(* IEC 61131-3 sources: SmartHomeNew/ (part 4) *)

(* ---- FB_Cluster_Runtime_FSM.st ---- *)
FUNCTION_BLOCK FB_Cluster_Runtime_FSM
VAR_INPUT
    VI_Enable : BOOL;
    VI_System_Time_MS : UDINT;
END_VAR

IF NOT VI_Enable THEN
    GVL_Cluster_Runtime_FSM.G_Runtime_Valid := FALSE;
    RETURN;
END_IF;

// Reset runtime states.
GVL_Cluster_Runtime_FSM.G_State_Startup := FALSE;
GVL_Cluster_Runtime_FSM.G_State_Discovery := FALSE;
GVL_Cluster_Runtime_FSM.G_State_Synchronization := FALSE;
GVL_Cluster_Runtime_FSM.G_State_Operational := FALSE;
GVL_Cluster_Runtime_FSM.G_State_Degraded := FALSE;
GVL_Cluster_Runtime_FSM.G_State_Observer_Only := FALSE;
GVL_Cluster_Runtime_FSM.G_State_Recovery_Lock := FALSE;
GVL_Cluster_Runtime_FSM.G_State_Quarantine := FALSE;

// Startup state.
IF NOT GVL_Distributed_Runtime.G_Runtime_Valid THEN

    GVL_Cluster_Runtime_FSM.G_State_Startup := TRUE;

    GVL_Cluster_Runtime_FSM.G_Status_Code := 1;
    GVL_Cluster_Runtime_FSM.G_Status_Text :=
        'Cluster runtime startup';

ELSIF GVL_Runtime_Discovery.G_Runtime_Valid
   AND NOT GVL_Runtime_Discovery.G_Any_Discovery_Rejected THEN

    GVL_Cluster_Runtime_FSM.G_State_Discovery := TRUE;

    GVL_Cluster_Runtime_FSM.G_Status_Code := 2;
    GVL_Cluster_Runtime_FSM.G_Status_Text :=
        'Cluster runtime discovery';

END_IF;

// Synchronization state.
IF GVL_Runtime_Bus.G_TX_Healthy
   AND GVL_Runtime_Bus.G_RX_Healthy THEN

    GVL_Cluster_Runtime_FSM.G_State_Synchronization := TRUE;

END_IF;

// Operational state.
IF GVL_Distributed_Execution_Gates.G_Can_Execute
   AND GVL_Distributed_Execution_Gates.G_Can_Orchestrate THEN

    GVL_Cluster_Runtime_FSM.G_State_Operational := TRUE;

    GVL_Cluster_Runtime_FSM.G_Status_Code := 0;
    GVL_Cluster_Runtime_FSM.G_Status_Text :=
        'Cluster runtime operational';

END_IF;

// Degraded state.
IF GVL_Cluster_Safety_Barrier.G_Cluster_Execution_Blocked THEN

    GVL_Cluster_Runtime_FSM.G_State_Degraded := TRUE;

    GVL_Cluster_Runtime_FSM.G_Status_Code := 10;
    GVL_Cluster_Runtime_FSM.G_Status_Text :=
        'Cluster runtime degraded';

END_IF;

// Observer-only state.
IF GVL_Distributed_Authority.G_Authority_State.Authority_Observer_Only THEN

    GVL_Cluster_Runtime_FSM.G_State_Observer_Only := TRUE;

    GVL_Cluster_Runtime_FSM.G_Status_Code := 11;
    GVL_Cluster_Runtime_FSM.G_Status_Text :=
        'Cluster runtime observer-only';

END_IF;

// Recovery lock state.
IF GVL_Distributed_Recovery_Lock.G_Recovery_Execution_Blocked THEN

    GVL_Cluster_Runtime_FSM.G_State_Recovery_Lock := TRUE;

    GVL_Cluster_Runtime_FSM.G_Status_Code := 12;
    GVL_Cluster_Runtime_FSM.G_Status_Text :=
        'Cluster runtime recovery-locked';

END_IF;

// Quarantine state.
IF GVL_Runtime_Discovery.G_Any_Node_Quarantined THEN

    GVL_Cluster_Runtime_FSM.G_State_Quarantine := TRUE;

    GVL_Cluster_Runtime_FSM.G_Status_Code := 13;
    GVL_Cluster_Runtime_FSM.G_Status_Text :=
        'Cluster runtime quarantined';

END_IF;

GVL_Cluster_Runtime_FSM.G_Runtime_Valid := TRUE;
GVL_Cluster_Runtime_FSM.G_Last_Update_MS := VI_System_Time_MS;

END_FUNCTION_BLOCK

(* ---- FB_Cluster_Safety_Barrier_Runtime.st ---- *)
FUNCTION_BLOCK FB_Cluster_Safety_Barrier_Runtime
VAR_INPUT
    VI_Enable : BOOL;
    VI_System_Time_MS : UDINT;
END_VAR
VAR
    L_Block_Execution : BOOL;
    L_Status_Code : UINT;
    L_Status_Text : STRING(160);
END_VAR

IF NOT VI_Enable THEN
    GVL_Cluster_Safety_Barrier.G_Runtime_Valid := FALSE;
    RETURN;
END_IF;

L_Block_Execution := FALSE;
L_Status_Code := 0;
L_Status_Text := 'Cluster safety barrier healthy';

GVL_Cluster_Safety_Barrier.G_Remote_Authority_Degraded := FALSE;
GVL_Cluster_Safety_Barrier.G_Runtime_Bus_Degraded := FALSE;
GVL_Cluster_Safety_Barrier.G_Projection_Ownership_Invalid := FALSE;
GVL_Cluster_Safety_Barrier.G_Recovery_Lock_Active := FALSE;
GVL_Cluster_Safety_Barrier.G_Deployment_Invalid := FALSE;
GVL_Cluster_Safety_Barrier.G_Authority_Downgraded := FALSE;
GVL_Cluster_Safety_Barrier.G_Orchestration_Restricted := FALSE;

// Remote authority staleness barrier.
IF GVL_Distributed_Runtime.G_Any_Remote_Node_Offline
   OR GVL_Distributed_Runtime.G_Split_Brain_Suspected THEN

    L_Block_Execution := TRUE;
    L_Status_Code := 10;
    L_Status_Text :=
        'Cluster authority state degraded';

    GVL_Cluster_Safety_Barrier.G_Remote_Authority_Degraded := TRUE;

END_IF;

// Runtime bus integrity barrier.
IF GVL_Runtime_Bus.G_Any_Replication_Rejected
   OR NOT GVL_Runtime_Bus.G_TX_Healthy
   OR NOT GVL_Runtime_Bus.G_RX_Healthy THEN

    L_Block_Execution := TRUE;
    L_Status_Code := 11;
    L_Status_Text :=
        'Runtime bus integrity degraded';

    GVL_Cluster_Safety_Barrier.G_Runtime_Bus_Degraded := TRUE;

END_IF;

// Projection ownership barrier.
IF GVL_Distributed_Projection_Ownership.G_Any_Ownership_Conflict
   OR GVL_Distributed_Projection_Ownership.G_Any_Ownership_Stale THEN

    L_Block_Execution := TRUE;
    L_Status_Code := 12;
    L_Status_Text :=
        'Distributed projection ownership invalid';

    GVL_Cluster_Safety_Barrier.G_Projection_Ownership_Invalid := TRUE;

END_IF;

// Recovery lock barrier.
IF GVL_Distributed_Recovery_Lock.G_Recovery_Execution_Blocked
   OR GVL_Distributed_Recovery_Lock.G_Rollback_Execution_Blocked
   OR GVL_Distributed_Recovery_Lock.G_Reopen_Execution_Blocked THEN

    L_Block_Execution := TRUE;
    L_Status_Code := 13;
    L_Status_Text :=
        'Distributed recovery execution blocked';

    GVL_Cluster_Safety_Barrier.G_Recovery_Lock_Active := TRUE;

END_IF;

// Discovery/deployment barrier.
IF GVL_Runtime_Discovery.G_Any_Discovery_Rejected
   OR GVL_Runtime_Discovery.G_Any_Node_Quarantined THEN

    L_Block_Execution := TRUE;
    L_Status_Code := 14;
    L_Status_Text :=
        'Runtime deployment/discovery invalid';

    GVL_Cluster_Safety_Barrier.G_Deployment_Invalid := TRUE;

END_IF;

// Cluster escalation semantics.
IF L_Block_Execution THEN

    GVL_Distributed_Authority.G_Authority_State.Authority_Observer_Only := TRUE;
    GVL_Distributed_Authority.G_Authority_State.Authority_Master_Elected := FALSE;

    GVL_Distributed_Orchestration.G_Distributed_Projection_Healthy := FALSE;

    GVL_Cluster_Safety_Barrier.G_Authority_Downgraded := TRUE;
    GVL_Cluster_Safety_Barrier.G_Orchestration_Restricted := TRUE;

END_IF;

GVL_Cluster_Safety_Barrier.G_Cluster_Execution_Blocked :=
    L_Block_Execution;

GVL_Cluster_Safety_Barrier.G_Runtime_Valid := TRUE;
GVL_Cluster_Safety_Barrier.G_Last_Update_MS := VI_System_Time_MS;
GVL_Cluster_Safety_Barrier.G_Status_Code := L_Status_Code;
GVL_Cluster_Safety_Barrier.G_Status_Text := L_Status_Text;

END_FUNCTION_BLOCK

(* ---- FB_CO_Detector.st ---- *)
FUNCTION_BLOCK FB_CO_Detector
VAR_INPUT
    VI_CO_PPM : REAL;
    VI_Threshold_Warning : REAL := 30.0;
    VI_Threshold_Alarm   : REAL := 70.0;
END_VAR
VAR_OUTPUT
    VO_CO_Warning_Level : BOOL;
    VO_CO_Alarm_Level   : BOOL;
END_VAR

VO_CO_Warning_Level := (VI_CO_PPM >= VI_Threshold_Warning);
VO_CO_Alarm_Level   := (VI_CO_PPM >= VI_Threshold_Alarm);

(* ---- FB_Command_Deduplication.st ---- *)
FUNCTION_BLOCK FB_Command_Deduplication
VAR_INPUT
    VI_Command_ID : UDINT; // Unique ID from Gateway/HMI
    VI_Command_Type : E_Gateway_Command_Type;
    VI_Command_Value : REAL;
    VI_System_Time_MS : UDINT;
END_VAR
VAR_OUTPUT
    VO_Is_New_Command : BOOL; // TRUE if this command should be executed
    VO_Processed_ID : UDINT;
END_VAR
VAR
    L_Processed_History : ARRAY[0..GVL_CONSTANTS.C_MAX_DEDUPLICATION_HISTORY-1] OF UDINT;
    L_Processed_Times   : ARRAY[0..GVL_CONSTANTS.C_MAX_DEDUPLICATION_HISTORY-1] OF UDINT;
    L_History_Index : INT := 0;
    L_i : INT;
    L_Found : BOOL;
    L_Age_MS : UDINT;
END_VAR

L_Found := FALSE;

FOR L_i := 0 TO GVL_CONSTANTS.C_MAX_DEDUPLICATION_HISTORY - 1 DO
    IF (L_Processed_History[L_i] = VI_Command_ID) AND (VI_Command_ID <> 0) THEN
        IF VI_System_Time_MS >= L_Processed_Times[L_i] THEN
            L_Age_MS := VI_System_Time_MS - L_Processed_Times[L_i];
        ELSE
            L_Age_MS := (4294967295 - L_Processed_Times[L_i]) + VI_System_Time_MS + 1;
        END_IF;

        IF L_Age_MS < 3600000 THEN
            L_Found := TRUE;
            EXIT;
        END_IF;
    END_IF;
END_FOR;

IF (NOT L_Found) AND (VI_Command_ID <> 0) THEN
    VO_Is_New_Command := TRUE;
    VO_Processed_ID := VI_Command_ID;

    L_Processed_History[L_History_Index] := VI_Command_ID;
    L_Processed_Times[L_History_Index] := VI_System_Time_MS;

    L_History_Index := L_History_Index + 1;
    IF L_History_Index > GVL_CONSTANTS.C_MAX_DEDUPLICATION_HISTORY - 1 THEN
        L_History_Index := 0;
    END_IF;
ELSE
    VO_Is_New_Command := FALSE;
    VO_Processed_ID := 0;
END_IF;
END_FUNCTION_BLOCK

(* ---- FB_Config_Activation_Runtime.st ---- *)
FUNCTION_BLOCK FB_Config_Activation_Runtime
VAR_INPUT
    VI_Enable : BOOL;
    VI_System_Time_MS : UDINT;
END_VAR
VAR
    L_i : INT;
    L_State : ST_Config_Activation_State;
    L_Staged_Valid : BOOL;
END_VAR

IF NOT VI_Enable THEN
    GVL_Config_Activation.G_Activation_Runtime_Valid := FALSE;
    RETURN;
END_IF;

L_State.Runtime_Valid := TRUE;
L_State.Runtime_System_Time_MS := VI_System_Time_MS;

L_State.Active_Version :=
    GVL_Water_Topology_Config.G_Active_Config_Version;

L_State.Staged_Version :=
    GVL_Config_Activation.G_Staged_Config_Version;

L_State.Previous_Stable_Version :=
    GVL_Config_Activation.G_Last_Stable_Config_Version;

L_State.Activation_Requested :=
    GVL_Config_Activation.G_Activation_Request;

L_State.Rollback_Requested :=
    GVL_Config_Activation.G_Rollback_Request;

L_State.Rollback_Available :=
    GVL_Config_Activation.G_Last_Stable_Config_Version <> 0;

L_Staged_Valid := TRUE;

FOR L_i := 1 TO GVL_CONSTANTS.C_MAX_FLOOD_SENSORS DO

    IF GVL_Config_Activation.G_Staged_Topology_Config[L_i].Primary_Valve_Group_Id = 0 THEN
        L_Staged_Valid := FALSE;
    END_IF;

END_FOR;

L_State.Staged_Config_Valid := L_Staged_Valid;
L_State.Migration_Compatible := TRUE;

IF L_State.Rollback_Requested THEN

    IF L_State.Rollback_Available THEN

        L_State.Rollback_Active := TRUE;
        L_State.Activation_Blocked := TRUE;

        GVL_Config_Activation.G_Config_Quarantine_Active := FALSE;

        L_State.Status_Code := 3;
        L_State.Status_Text := 'Rollback activation active';

    ELSE

        L_State.Rollback_Active := FALSE;
        L_State.Activation_Blocked := TRUE;

        L_State.Status_Code := 4;
        L_State.Status_Text := 'Rollback rejected: no stable version';

    END_IF;

    GVL_Config_Activation.G_Rollback_Request := FALSE;

ELSIF L_State.Activation_Requested THEN

    IF NOT L_State.Staged_Config_Valid THEN

        L_State.Activation_Blocked := TRUE;
        L_State.Config_Quarantine_Active := TRUE;

        GVL_Config_Activation.G_Config_Quarantine_Active := TRUE;

        L_State.Status_Code := 2;
        L_State.Status_Text := 'Config activation quarantined';

    ELSE

        L_State.Activation_Allowed := TRUE;

        GVL_Water_Topology_Config_Source.G_Source_Version :=
            L_State.Staged_Version;

        FOR L_i := 1 TO GVL_CONSTANTS.C_MAX_FLOOD_SENSORS DO

            GVL_Water_Topology_Config_Source.G_Source_Record[L_i] :=
                GVL_Config_Activation.G_Staged_Topology_Config[L_i];

        END_FOR;

        GVL_Water_Topology_Config_Source.G_Source_Valid := TRUE;
        GVL_Water_Topology_Config_Source.G_Source_Activated_MS := VI_System_Time_MS;

        GVL_Config_Activation.G_Last_Stable_Config_Version :=
            L_State.Staged_Version;

        GVL_Config_Activation.G_Config_Quarantine_Active := FALSE;

        L_State.Status_Code := 1;
        L_State.Status_Text := 'Config activation completed';

    END_IF;

    GVL_Config_Activation.G_Activation_Request := FALSE;

ELSE

    L_State.Status_Code := 0;
    L_State.Status_Text := 'Config activation runtime healthy';

END_IF;

GVL_Config_Activation.G_Activation_State := L_State;

GVL_Config_Activation.G_Activation_Runtime_Valid := TRUE;
GVL_Config_Activation.G_Last_Update_MS := VI_System_Time_MS;
GVL_Config_Activation.G_Status_Code := L_State.Status_Code;
GVL_Config_Activation.G_Status_Text := L_State.Status_Text;

END_FUNCTION_BLOCK

(* ---- FB_Config_Simulation.st ---- *)
// ==============================================================================
// Config simulation / validation function block
// Service/commissioning validation utility.
// Does NOT own runtime control and does NOT participate in heating phase runtime.
// ==============================================================================
FUNCTION_BLOCK FB_Config_Simulation
VAR_INPUT
    VI_Enable : BOOL;
    VI_Request : BOOL;
    VI_Confirm : BOOL;
END_VAR
VAR_OUTPUT
    VO_Executed : BOOL;
    VO_Result_OK : BOOL;
    VO_Error_Text : STRING(200);
END_VAR
VAR
    L_Error : BOOL;
END_VAR

VO_Executed := FALSE;
VO_Result_OK := GVL_CONFIG_SIMULATION.G_Simulation_Result_OK;
VO_Error_Text := GVL_CONFIG_SIMULATION.G_Simulation_Error_Text;

IF NOT VI_Enable THEN
    RETURN;
END_IF;

IF VI_Request AND VI_Confirm THEN

    L_Error := FALSE;
    VO_Result_OK := TRUE;
    VO_Error_Text := '';

    // Simulate INPUT constraints.
    IF (GVL_CONFIG_CONTROL.STG_Reputation_Learning_Rate < 0.0) OR (GVL_CONFIG_CONTROL.STG_Reputation_Learning_Rate > 1.0) THEN
        VO_Result_OK := FALSE;
        VO_Error_Text := 'Invalid learning rate';
        L_Error := TRUE;
    END_IF;

    IF (GVL_CONFIG_CONTROL.STG_Reputation_Recovery_Decay < 0.0) OR (GVL_CONFIG_CONTROL.STG_Reputation_Recovery_Decay > 1.0) THEN
        VO_Result_OK := FALSE;
        VO_Error_Text := 'Invalid recovery decay';
        L_Error := TRUE;
    END_IF;

    IF (GVL_CONFIG_CONTROL.STG_Min_Sensor_Confidence < 0.0) OR (GVL_CONFIG_CONTROL.STG_Min_Sensor_Confidence > 1.0) THEN
        VO_Result_OK := FALSE;
        VO_Error_Text := 'Invalid minimum confidence';
        L_Error := TRUE;
    END_IF;

    IF (GVL_CONFIG_CONTROL.STG_Bad_Spike_Confidence < 0.0) OR (GVL_CONFIG_CONTROL.STG_Bad_Spike_Confidence > 1.0) THEN
        VO_Result_OK := FALSE;
        VO_Error_Text := 'Invalid spike confidence';
        L_Error := TRUE;
    END_IF;

    IF (GVL_CONFIG_CONTROL.STG_Default_Confidence < 0.0) OR (GVL_CONFIG_CONTROL.STG_Default_Confidence > 1.0) THEN
        VO_Result_OK := FALSE;
        VO_Error_Text := 'Invalid default confidence';
        L_Error := TRUE;
    END_IF;

    // Simulate SCENARIO logic.
    IF (GVL_CONFIG_CONTROL.STG_Night_Start_Hour < 0) OR (GVL_CONFIG_CONTROL.STG_Night_Start_Hour > 23) THEN
        VO_Result_OK := FALSE;
        VO_Error_Text := 'Night start hour invalid';
        L_Error := TRUE;
    END_IF;

    IF (GVL_CONFIG_CONTROL.STG_Night_End_Hour < 0) OR (GVL_CONFIG_CONTROL.STG_Night_End_Hour > 23) THEN
        VO_Result_OK := FALSE;
        VO_Error_Text := 'Night end hour invalid';
        L_Error := TRUE;
    END_IF;

    IF GVL_CONFIG_CONTROL.STG_Night_Start_Hour = GVL_CONFIG_CONTROL.STG_Night_End_Hour THEN
        VO_Result_OK := FALSE;
        VO_Error_Text := 'Night window invalid';
        L_Error := TRUE;
    END_IF;

    IF (GVL_CONFIG_CONTROL.STG_VentBoost_Humidity_Threshold < 0.0) OR (GVL_CONFIG_CONTROL.STG_VentBoost_Humidity_Threshold > 100.0) THEN
        VO_Result_OK := FALSE;
        VO_Error_Text := 'Humidity threshold invalid';
        L_Error := TRUE;
    END_IF;

    // Simulate SAFETY.
    IF GVL_CONFIG_CONTROL.STG_Stabilization_Delay_MS < 1000 THEN
        VO_Result_OK := FALSE;
        VO_Error_Text := 'Recovery delay too small';
        L_Error := TRUE;
    END_IF;

    // Simulate FAIL-SAFE policy.
    IF NOT (
        GVL_CONFIG_CONTROL.STG_PLC_Inactive_Close_Gas OR
        GVL_CONFIG_CONTROL.STG_PLC_Inactive_Stop_Boiler OR
        GVL_CONFIG_CONTROL.STG_PLC_Inactive_Block_Heating OR
        GVL_CONFIG_CONTROL.STG_PLC_Inactive_Stop_Vent OR
        GVL_CONFIG_CONTROL.STG_PLC_Inactive_Block_Water
    ) THEN
        VO_Result_OK := FALSE;
        VO_Error_Text := 'Fail-safe disabled';
        L_Error := TRUE;
    END_IF;

    GVL_CONFIG_SIMULATION.G_Simulation_Result_OK := NOT L_Error;
    GVL_CONFIG_SIMULATION.G_Simulation_Error_Text := VO_Error_Text;
    GVL_CONFIG_SIMULATION.G_Simulation_Last_Run_MS := GVL_TIME_SERVICE.G_Now_MS;
    GVL_CONFIG_SIMULATION.G_Simulation_Result_Seq := GVL_CONFIG_SIMULATION.G_Simulation_Result_Seq + 1;
    GVL_CONFIG_SIMULATION.G_Simulation_Staged_Config_Version := GVL_CONFIG_CONTROL.G_Staged_Config_Version;
    VO_Executed := TRUE;

    // One-shot request consumption. HMI/service callers get the result from
    // GVL_CONFIG_SIMULATION and must raise a new request for another run.
    GVL_CONFIG_SIMULATION.G_Simulation_Request := FALSE;
    GVL_CONFIG_SIMULATION.G_Simulation_Confirm := FALSE;

END_IF;

END_FUNCTION_BLOCK
// >>> BULK_SYNC_ANCHOR: FB_Config_Simulation <<<

(* ---- FB_CoreKernel_Live_Observer.st ---- *)
FUNCTION_BLOCK FB_CoreKernel_Live_Observer
END_FUNCTION_BLOCK

(* ---- FB_DHW_Manager.st ---- *)
FUNCTION_BLOCK FB_DHW_Manager
VAR_INPUT
    VI_System_Time_MS : UDINT; // Системное время (мс)
    VI_Current_TOD : TOD; // Текущее время суток
    VI_IsActivePLC : BOOL; // Флаг: Данный ПЛК является ведущим
    VI_Temp : REAL; // Текущая температура воды в бойлере (°C)
    VI_Pressure : REAL; // Текущее давление в системе ГВС (бар)
    VI_Config : ST_DHW_Config; // Конфигурация системы ГВС (уставки, расписание)
    VI_Current_Day_Of_Week : UINT; // Текущий день недели (1-7)
    VI_Reset_Errors : BOOL; // Сброс ошибок
    VI_Emergency_Stop : BOOL; // Агрегированный аварийный стоп от подсистемы безопасности
    VI_System_Mode : E_System_Operating_Mode; // Агрегированный режим системы
    VI_IO_Modules_Online : ARRAY[1..GVL_CONSTANTS.C_MAX_MODULES] OF BOOL; // Статусы модулей ввода-вывода (только чтение)
END_VAR
// >>> SYNC_TEST_MARKER_001 <<<
VAR_OUTPUT
    VO_Status : ST_DHW_Status; // Сводный статус системы ГВС для HMI
    VO_Heating_Pump : BOOL; // Выход: Управление насосом нагрева (загрузка бойлера)
    VO_Circ_Pump : BOOL; // Выход: Управление насосом рециркуляции ГВС
END_VAR
VAR
    // DHW V2 staging layer
    L_DHW_V2_Command_V2 : ST_DHW_Command_V2;
    L_DHW_V2_State_V2 : ST_DHW_State_V2;
    L_DHW_V2_Shadow_Diff_Found : BOOL;
    L_DHW_V2_Switch_Enabled : BOOL;
    L_DHW_V2_Path_Ready : BOOL;
    L_DHW_Using_Legacy_Fallback : BOOL;
    L_i : INT;
    L_Current_TOD : TOD; // Текущее время суток
    L_Legionella_Active : BOOL; // Флаг активного режима термической дезинфекции (Легионелла)
    L_Legionella_Timer : FB_System_Timer; // Таймер удержания температуры для дезинфекции
    L_Last_Good_Temp : REAL := 55.0; // Последнее достоверное значение температуры (для Fallback)
    L_Legionella_Done_Today : BOOL; // Признак выполнения термодезинфекции в текущие сутки
    L_Last_Legionella_Day : UINT; // День недели последнего сброса/контроля цикла легионеллы
    fbTempValidator : FB_Analog_Validator;
    fbPressValidator : FB_Analog_Validator;
    L_Error_Latched : BOOL;
    L_Error_ID_Latched : WORD;
    L_Policy_Degraded : BOOL;
    L_Policy_Freeze_Protection : BOOL;
    L_Policy_Safe_Stop : BOOL;
    L_Target_Temp_Adjusted : REAL;
END_VAR

IF NOT VI_IsActivePLC THEN RETURN; END_IF;

L_DHW_V2_Shadow_Diff_Found := FALSE;
L_DHW_V2_Switch_Enabled := TRUE;
L_DHW_V2_Path_Ready := FALSE;
L_DHW_Using_Legacy_Fallback := TRUE;

GVL_STATE.G_DHW_IO_Fault := FALSE;
GVL_STATE.G_DHW_Sensor_Fault := FALSE;
GVL_STATE.G_DHW_Subsystem_Degraded := FALSE;

IF VI_Emergency_Stop THEN
    VO_Heating_Pump := FALSE;
    VO_Circ_Pump := FALSE;
    VO_Status.Warning := FALSE;
    VO_Status.Error := TRUE;
    VO_Status.Error_ID := TO_WORD(GVL_CONFIG.ERR_DHW_IO_OFFLINE); // временно используем общий аварийный код до детализации safety-кодов
    VO_Status.Heating_Pump_On := FALSE;
    VO_Status.Circ_Pump_On := FALSE;
    RETURN;
END_IF;

// Фиксация текущего времени
L_Current_TOD := VI_Current_TOD;

// ========================================
// DHW POLICY LAYER
// ========================================
L_Policy_Safe_Stop := (VI_System_Mode = E_System_Operating_Mode.MODE_SAFE_STOP);
L_Policy_Freeze_Protection := (VI_System_Mode = E_System_Operating_Mode.MODE_FREEZE_PROTECTION);
L_Policy_Degraded := (VI_System_Mode = E_System_Operating_Mode.MODE_DEGRADED);
L_Target_Temp_Adjusted := VI_Config.Target_Temp;
IF L_Policy_Degraded THEN
    L_Target_Temp_Adjusted := VI_Config.Target_Temp - VI_Config.Degraded_Target_Delta;
END_IF;

// ========================================
// DHW POLICY OVERRIDE
// ========================================
IF L_Policy_Safe_Stop THEN
    VO_Heating_Pump := FALSE;
    VO_Circ_Pump := FALSE;
    RETURN;
END_IF;

IF L_Policy_Freeze_Protection THEN
    VO_Heating_Pump := FALSE;
    VO_Circ_Pump := FALSE;
    RETURN;
END_IF;

// Сброс признака выполнения термодезинфекции при смене дня.
IF L_Last_Legionella_Day <> VI_Current_Day_Of_Week THEN
    L_Legionella_Done_Today := FALSE;
    L_Last_Legionella_Day := VI_Current_Day_Of_Week;
END_IF;

// Базовый сброс незащёлкнутых статусных флагов на текущий цикл.
// Критические ошибки ниже могут зафиксироваться и завершить выполнение через RETURN.
VO_Status.Warning := FALSE;
VO_Status.Error := FALSE;
VO_Status.Error_ID := 0;

// Сброс ошибок
IF VI_Reset_Errors THEN
    L_Error_Latched := FALSE;
    L_Error_ID_Latched := 0;
END_IF;

// Проверка связи с модулями ввода-вывода
FOR L_i := 1 TO GVL_CONSTANTS.C_MAX_MODULES DO
    IF NOT VI_IO_Modules_Online[L_i] THEN
        L_Error_Latched := TRUE;
        GVL_STATE.G_DHW_IO_Fault := TRUE;
        L_Error_ID_Latched := TO_WORD(GVL_CONFIG.ERR_DHW_IO_OFFLINE); // Потеря связи с модулями ввода-вывода
    END_IF;
END_FOR;

// 1. Обработка неисправностей датчиков и сервисных режимов (ТЗ 7.0)
fbTempValidator(
    VI_Value := VI_Temp,
    VI_Min_Valid := 0.0,
    VI_Max_Valid := 100.0,
    VI_Fallback_Mode := 0,
    VI_Default_Value := 55.0
);

fbPressValidator(
    VI_Value := VI_Pressure,
    VI_Min_Valid := 0.0,
    VI_Max_Valid := 10.0,
    VI_Fallback_Mode := 0
);

VO_Status.Temp := fbTempValidator.VO_Value;
VO_Status.Pressure := fbPressValidator.VO_Value;

// Сохраняем последнее достоверное значение температуры ГВС.
// Используется только для диагностики/сервиса, не для fallback-управления.
IF NOT fbTempValidator.VO_Error THEN
    L_Last_Good_Temp := VO_Status.Temp;
END_IF;

IF fbTempValidator.VO_Error THEN
    GVL_STATE.G_DHW_Sensor_Fault := TRUE;
    L_Error_Latched := TRUE;
    L_Error_ID_Latched := TO_WORD(GVL_CONFIG.ERR_DHW_TEMP_SENSOR_FAULT); // Критическая ошибка датчика температуры
ELSIF (VO_Status.Pressure < 1.0 OR VO_Status.Pressure > 4.0) AND NOT fbPressValidator.VO_Error THEN
    L_Error_Latched := TRUE;
    L_Error_ID_Latched := TO_WORD(GVL_CONFIG.ERR_DHW_PRESSURE_OUT_OF_RANGE); // Давление вне нормы
END_IF;

IF L_Error_Latched THEN
    // Критическая ошибка: переход в безопасное состояние с полной остановкой насосов.
    VO_Heating_Pump := FALSE;
    VO_Circ_Pump := FALSE;
    VO_Status.Warning := FALSE;
    VO_Status.Error := TRUE;
    VO_Status.Error_ID := L_Error_ID_Latched;
    VO_Status.Heating_Pump_On := FALSE;
    VO_Status.Circ_Pump_On := FALSE;
    RETURN;
END_IF;

// Ошибка датчика давления не останавливает ГВС,
// но переводит подсистему в режим предупреждения (degraded mode).
IF fbPressValidator.VO_Error THEN
    GVL_STATE.G_DHW_Sensor_Fault := TRUE;
    GVL_STATE.G_DHW_Subsystem_Degraded := TRUE;
    VO_Status.Warning := TRUE;
    VO_Status.Error := FALSE;
    VO_Status.Error_ID := TO_WORD(GVL_CONFIG.ERR_DHW_PRESSURE_SENSOR_FAULT);
END_IF;

// 2. Логика поддержания температуры воды в бойлере (Нагрев)
// На этом этапе FB уже выполняется только на активном ПЛК.

// Термическая дезинфекция (Легионелла)
IF VI_Config.Anti_Legionella_Enabled
   AND (VI_Current_Day_Of_Week = VI_Config.Anti_Legionella_Day)
   AND (L_Current_TOD >= TOD#02:00)
   AND (L_Current_TOD <= TOD#04:00)
   AND NOT L_Legionella_Done_Today THEN
    L_Legionella_Active := TRUE;
ELSE
    L_Legionella_Active := FALSE;
END_IF;

L_Legionella_Timer(IN := L_Legionella_Active AND VO_Status.Temp >= 70.0, PT := T#30m, VI_System_Time_MS := VI_System_Time_MS);
IF L_Legionella_Timer.Q THEN
    L_Legionella_Active := FALSE; // Дезинфекция завершена
    L_Legionella_Done_Today := TRUE; // Повторно в те же сутки не запускать
END_IF;

// Двухпозиционное регулирование с гистерезисом
IF L_Legionella_Active THEN
    IF VO_Status.Temp < 70.0 THEN
        VO_Heating_Pump := TRUE;
    ELSIF VO_Status.Temp > 72.0 THEN
        VO_Heating_Pump := FALSE;
    END_IF;
ELSE
    IF VO_Status.Temp < (L_Target_Temp_Adjusted - VI_Config.Hysteresis) THEN
        VO_Heating_Pump := TRUE;
    ELSIF VO_Status.Temp > (L_Target_Temp_Adjusted + VI_Config.Hysteresis) THEN
        VO_Heating_Pump := FALSE;
    END_IF;
END_IF;

// 3. Управление циркуляционным насосом ГВС по расписанию
// Рециркуляция обеспечивает мгновенное наличие горячей воды у потребителя
VO_Circ_Pump := SEL(VI_Config.Circulation_Schedule_Enabled AND NOT (VI_Config.Night_Mode_Enabled AND (L_Current_TOD < VI_Config.Circulation_Start OR L_Current_TOD > VI_Config.Circulation_End)), FALSE, TRUE);

// Формирование статусных данных для визуализации.
// К этому моменту статус уже консистентен:
// - Error = критическая ошибка с остановкой ГВС
// - Warning = деградация без остановки
VO_Status.Heating_Pump_On := VO_Heating_Pump;
VO_Status.Circ_Pump_On := VO_Circ_Pump;

// ========================================
// DHW V2 shadow execution (phase2)
// Inlined from FB_DHW_V2_Staging
// ========================================
IF VO_Heating_Pump THEN
    L_DHW_V2_Command_V2.Pump_Enable := 1.0;
ELSE
    L_DHW_V2_Command_V2.Pump_Enable := 0.0;
END_IF;

L_DHW_V2_State_V2.Tank_Temp := VO_Status.Temp;
L_DHW_V2_State_V2.Supply_Temp := VO_Status.Pressure;

// ========================================
// DHW V2 staging validation
// ========================================
IF VO_Heating_Pump <> (L_DHW_V2_Command_V2.Pump_Enable > 0.5) THEN
    L_DHW_V2_Shadow_Diff_Found := TRUE;
END_IF;
IF ABS(VO_Status.Temp - L_DHW_V2_State_V2.Tank_Temp) > 0.1 THEN
    L_DHW_V2_Shadow_Diff_Found := TRUE;
END_IF;
IF ABS(VO_Status.Pressure - L_DHW_V2_State_V2.Supply_Temp) > 0.1 THEN
    L_DHW_V2_Shadow_Diff_Found := TRUE;
END_IF;

// Guarded DHW V2 enable
IF L_DHW_V2_Switch_Enabled THEN
    IF NOT L_DHW_V2_Shadow_Diff_Found THEN
        L_DHW_V2_Path_Ready := TRUE;
        L_DHW_Using_Legacy_Fallback := FALSE;
    ELSE
        L_DHW_V2_Path_Ready := FALSE;
        L_DHW_Using_Legacy_Fallback := TRUE;
    END_IF;
ELSE
    L_DHW_V2_Path_Ready := FALSE;
    L_DHW_Using_Legacy_Fallback := TRUE;
END_IF;

END_FUNCTION_BLOCK
// >>> BULK_SYNC_ANCHOR: FB_DHW_Manager <<<

(* ---- FB_Diagnostics_Event_Manager.st ---- *)
FUNCTION_BLOCK FB_Diagnostics_Event_Manager
VAR_INPUT
    VI_Code : UDINT;
    VI_Severity : INT;
    VI_Active : BOOL;
    VI_Timestamp : UDINT;
    VI_Source : INT;
END_VAR
VAR_IN_OUT
    VIO_Events : ARRAY[1..50] OF ST_Diagnostic_Event;
    VIO_Count : INT;
END_VAR
VAR
    L_Index : INT;
    L_i : INT;
    L_Found_Index : INT;
    L_Was_Active : BOOL;
    L_Debounce_Index : INT;
    L_Free_Debounce_Index : INT;
    L_Stable_State : BOOL;

    // Per-event anti-flapping state, keyed by (Code, Source)
    L_Debounce_Used : ARRAY[1..50] OF BOOL;
    L_Debounce_Code : ARRAY[1..50] OF UDINT;
    L_Debounce_Source : ARRAY[1..50] OF INT;
    L_Debounce_Last_Input_State : ARRAY[1..50] OF BOOL;
    L_Debounce_Stable_State : ARRAY[1..50] OF BOOL;
    L_Debounce_Last_Change_Time : ARRAY[1..50] OF UDINT;
END_VAR

// ======================================================
// FIND EXISTING EVENT
// ======================================================
L_Found_Index := 0;
L_Was_Active := FALSE;

FOR L_i := 1 TO 50 DO
    IF (VIO_Events[L_i].Code = VI_Code) AND (VIO_Events[L_i].Source = VI_Source) THEN
        L_Found_Index := L_i;
        L_Was_Active := VIO_Events[L_i].Active;
        EXIT;
    END_IF;
END_FOR;

// ======================================================
// FIND / ALLOCATE PER-EVENT DEBOUNCE SLOT
// ======================================================
L_Debounce_Index := 0;
L_Free_Debounce_Index := 0;

FOR L_i := 1 TO 50 DO
    IF L_Debounce_Used[L_i] THEN
        IF (L_Debounce_Code[L_i] = VI_Code) AND (L_Debounce_Source[L_i] = VI_Source) THEN
            L_Debounce_Index := L_i;
            EXIT;
        END_IF;
    ELSIF L_Free_Debounce_Index = 0 THEN
        L_Free_Debounce_Index := L_i;
    END_IF;
END_FOR;

IF L_Debounce_Index = 0 THEN
    IF L_Free_Debounce_Index > 0 THEN
        L_Debounce_Index := L_Free_Debounce_Index;
    ELSE
        // Deterministic fallback if debounce table is full.
        L_Debounce_Index := (VIO_Count MOD 50) + 1;
    END_IF;

    L_Debounce_Used[L_Debounce_Index] := TRUE;
    L_Debounce_Code[L_Debounce_Index] := VI_Code;
    L_Debounce_Source[L_Debounce_Index] := VI_Source;
    L_Debounce_Last_Input_State[L_Debounce_Index] := VI_Active;
    L_Debounce_Stable_State[L_Debounce_Index] := FALSE;
    L_Debounce_Last_Change_Time[L_Debounce_Index] := VI_Timestamp;
END_IF;

// ======================================================
// PER-EVENT ANTI-FLAPPING (2s debounce)
// ======================================================
IF VI_Active <> L_Debounce_Last_Input_State[L_Debounce_Index] THEN
    L_Debounce_Last_Input_State[L_Debounce_Index] := VI_Active;
    L_Debounce_Last_Change_Time[L_Debounce_Index] := VI_Timestamp;
END_IF;

IF (VI_Timestamp - L_Debounce_Last_Change_Time[L_Debounce_Index]) > 2000 THEN
    L_Debounce_Stable_State[L_Debounce_Index] := L_Debounce_Last_Input_State[L_Debounce_Index];
END_IF;

L_Stable_State := L_Debounce_Stable_State[L_Debounce_Index];

// ======================================================
// APPLY ONLY STABLE STATE
// ======================================================
IF L_Stable_State THEN
    IF NOT L_Was_Active THEN
        L_Index := (VIO_Count MOD 50) + 1;
        VIO_Events[L_Index].Code := VI_Code;
        VIO_Events[L_Index].Severity := VI_Severity;
        VIO_Events[L_Index].Active := TRUE;
        VIO_Events[L_Index].Timestamp := VI_Timestamp;
        VIO_Events[L_Index].Source := VI_Source;
        VIO_Count := VIO_Count + 1;
    ELSIF L_Found_Index > 0 THEN
        VIO_Events[L_Found_Index].Severity := VI_Severity;
    END_IF;
ELSE
    IF L_Found_Index > 0 THEN
        VIO_Events[L_Found_Index].Active := FALSE;
    END_IF;
END_IF;

// >>> BULK_SYNC_ANCHOR: FB_Diagnostics_Event_Manager <<<

(* ---- FB_Diagnostics_RootCause.st ---- *)
// ==============================================================================
// Heating root-cause inference engine
// Internal diagnostics core.
// Does NOT own explainability publication or runtime control.
// ==============================================================================
FUNCTION_BLOCK FB_Diagnostics_RootCause
VAR_INPUT
    // Safety / global blocking
    VI_Emergency_Stop : BOOL;
    VI_Gas_Safety : BOOL;
    VI_IO_Failsafe : BOOL;

    // Modern cascade semantic state
    VI_Cascade_Available : BOOL;
    VI_Cascade_Degraded : BOOL;
    VI_Cascade_Partial_Capacity : BOOL;
    VI_Cascade_No_Flame : BOOL;
    VI_Cascade_Transport_Degraded : BOOL;
    VI_Cascade_Ignition_Timeout : BOOL;
    VI_Cascade_Active_Boilers : UINT;
    VI_Cascade_Available_Boilers : UINT;

    // Boiler / OpenTherm state
    VI_Boiler_OT_Online : ARRAY[1..GVL_CONSTANTS.C_MAX_BOILERS] OF BOOL;
    VI_Boiler_Error : ARRAY[1..GVL_CONSTANTS.C_MAX_BOILERS] OF BOOL;
    VI_Boiler_Flame : ARRAY[1..GVL_CONSTANTS.C_MAX_BOILERS] OF BOOL;
    VI_Boiler_OT_Command_Timeout : ARRAY[1..GVL_CONSTANTS.C_MAX_BOILERS] OF BOOL;
    VI_Boiler_OT_Heartbeat_Timeout : ARRAY[1..GVL_CONSTANTS.C_MAX_BOILERS] OF BOOL;
    VI_Boiler_OT_Adapter_Error : ARRAY[1..GVL_CONSTANTS.C_MAX_BOILERS] OF BOOL;

    // Hydraulics
    VI_Manifold_Pumps : ARRAY[1..GVL_CONSTANTS.C_MAX_MANIFOLDS] OF BOOL;
    VI_Manifold_Valves : ARRAY[1..GVL_CONSTANTS.C_MAX_MANIFOLDS] OF REAL;

    // Sensors / thermal transfer
    VI_Sensor_Error : BOOL;
    VI_Supply_Temps : ARRAY[1..GVL_CONSTANTS.C_MAX_MANIFOLDS] OF REAL;
    VI_Target_Supply : REAL;
    VI_Demand_Map : ARRAY[1..GVL_CONSTANTS.C_MAX_MANIFOLDS] OF BOOL;
END_VAR

VAR_OUTPUT
    VO_RootCause : E_Heating_RootCause;
    VO_Confidence : REAL;
    VO_Error_Score : REAL;
    VO_Reason_Code : INT;
    VO_Reason_Text : STRING(128);
END_VAR

VAR
    L_i : INT;
    L_AnyBoilerOnline : BOOL;
    L_AnyBoilerError : BOOL;
    L_AnyFlame : BOOL;
    L_AnyCommandTimeout : BOOL;
    L_AnyHeartbeatTimeout : BOOL;
    L_AnyAdapterError : BOOL;
    L_AnyDemand : BOOL;
    L_AnyPumpOn : BOOL;
    L_AnyValveOpen : BOOL;
    L_LowSupply : BOOL;
    L_CascadeSemanticKnown : BOOL;
END_VAR

// ======================================================
// DEFAULTS
// ======================================================
VO_RootCause := E_Heating_RootCause.RC_NONE;
VO_Confidence := 1.0;
VO_Error_Score := 0.0;
VO_Reason_Code := 0;
VO_Reason_Text := 'Heating inference OK';

// ======================================================
// SAFETY / GLOBAL BLOCKS
// ======================================================
IF VI_Emergency_Stop THEN
    VO_RootCause := E_Heating_RootCause.RC_EMERGENCY_STOP;
    VO_Confidence := 1.0;
    VO_Error_Score := 1.0;
    VO_Reason_Code := 10;
    VO_Reason_Text := 'Emergency stop active';
    RETURN;
END_IF;

IF VI_Gas_Safety THEN
    VO_RootCause := E_Heating_RootCause.RC_GAS_SAFETY;
    VO_Confidence := 1.0;
    VO_Error_Score := 1.0;
    VO_Reason_Code := 20;
    VO_Reason_Text := 'Gas safety active';
    RETURN;
END_IF;

IF VI_IO_Failsafe THEN
    VO_RootCause := E_Heating_RootCause.RC_IO_OFFLINE;
    VO_Confidence := 1.0;
    VO_Error_Score := 1.0;
    VO_Reason_Code := 30;
    VO_Reason_Text := 'Heating IO failsafe active';
    RETURN;
END_IF;

// ======================================================
// AGGREGATE LEGACY / LOW-LEVEL FLAGS
// ======================================================
L_AnyBoilerOnline := FALSE;
L_AnyBoilerError := FALSE;
L_AnyFlame := FALSE;
L_AnyCommandTimeout := FALSE;
L_AnyHeartbeatTimeout := FALSE;
L_AnyAdapterError := FALSE;

FOR L_i := 1 TO GVL_CONSTANTS.C_MAX_BOILERS DO
    IF VI_Boiler_OT_Online[L_i] THEN
        L_AnyBoilerOnline := TRUE;
    END_IF;

    IF VI_Boiler_Error[L_i] THEN
        L_AnyBoilerError := TRUE;
    END_IF;

    IF VI_Boiler_Flame[L_i] THEN
        L_AnyFlame := TRUE;
    END_IF;

    IF VI_Boiler_OT_Command_Timeout[L_i] THEN
        L_AnyCommandTimeout := TRUE;
    END_IF;

    IF VI_Boiler_OT_Heartbeat_Timeout[L_i] THEN
        L_AnyHeartbeatTimeout := TRUE;
    END_IF;

    IF VI_Boiler_OT_Adapter_Error[L_i] THEN
        L_AnyAdapterError := TRUE;
    END_IF;
END_FOR;

L_AnyDemand := FALSE;
L_AnyPumpOn := FALSE;
L_AnyValveOpen := FALSE;
L_LowSupply := FALSE;

FOR L_i := 1 TO GVL_CONSTANTS.C_MAX_MANIFOLDS DO
    IF VI_Demand_Map[L_i] THEN
        L_AnyDemand := TRUE;
    END_IF;

    IF VI_Manifold_Pumps[L_i] THEN
        L_AnyPumpOn := TRUE;
    END_IF;

    IF VI_Manifold_Valves[L_i] > 5.0 THEN
        L_AnyValveOpen := TRUE;
    END_IF;

    IF VI_Demand_Map[L_i] AND (VI_Supply_Temps[L_i] < (VI_Target_Supply - 2.0)) THEN
        L_LowSupply := TRUE;
    END_IF;
END_FOR;

L_CascadeSemanticKnown :=
    VI_Cascade_Available OR
    VI_Cascade_Degraded OR
    VI_Cascade_Partial_Capacity OR
    VI_Cascade_No_Flame OR
    VI_Cascade_Transport_Degraded OR
    VI_Cascade_Ignition_Timeout OR
    (VI_Cascade_Active_Boilers > 0) OR
    (VI_Cascade_Available_Boilers > 0);

// ======================================================
// MODERN CASCADE / OPENTHERM SEMANTICS
// ======================================================
IF L_CascadeSemanticKnown THEN

    IF NOT VI_Cascade_Available THEN
        VO_RootCause := E_Heating_RootCause.RC_BOILER_OFFLINE;
        VO_Confidence := 0.95;
        VO_Error_Score := 0.95;
        VO_Reason_Code := 100;
        VO_Reason_Text := 'Heating cascade unavailable';
        RETURN;
    END_IF;

    IF VI_Cascade_Transport_Degraded THEN
        IF L_AnyHeartbeatTimeout THEN
            VO_RootCause := E_Heating_RootCause.RC_IO_OFFLINE;
            VO_Confidence := 0.90;
            VO_Error_Score := 0.90;
            VO_Reason_Code := 210;
            VO_Reason_Text := 'OpenTherm heartbeat timeout';
            RETURN;
        END_IF;

        IF L_AnyCommandTimeout THEN
            VO_RootCause := E_Heating_RootCause.RC_IO_OFFLINE;
            VO_Confidence := 0.85;
            VO_Error_Score := 0.85;
            VO_Reason_Code := 220;
            VO_Reason_Text := 'OpenTherm command ACK timeout';
            RETURN;
        END_IF;

        IF L_AnyAdapterError THEN
            VO_RootCause := E_Heating_RootCause.RC_IO_OFFLINE;
            VO_Confidence := 0.85;
            VO_Error_Score := 0.85;
            VO_Reason_Code := 230;
            VO_Reason_Text := 'OpenTherm adapter error';
            RETURN;
        END_IF;

        VO_RootCause := E_Heating_RootCause.RC_IO_OFFLINE;
        VO_Confidence := 0.75;
        VO_Error_Score := 0.75;
        VO_Reason_Code := 200;
        VO_Reason_Text := 'OpenTherm transport degraded';
        RETURN;
    END_IF;

    IF VI_Cascade_Ignition_Timeout THEN
        VO_RootCause := E_Heating_RootCause.RC_NO_FLAME;
        VO_Confidence := 0.90;
        VO_Error_Score := 0.90;
        VO_Reason_Code := 300;
        VO_Reason_Text := 'Boiler ignition timeout';
        RETURN;
    END_IF;

    IF VI_Cascade_No_Flame THEN
        VO_RootCause := E_Heating_RootCause.RC_NO_FLAME;
        VO_Confidence := 0.80;
        VO_Error_Score := 0.80;
        VO_Reason_Code := 310;
        VO_Reason_Text := 'Cascade active but no flame';
        RETURN;
    END_IF;

    IF VI_Cascade_Partial_Capacity THEN
        VO_RootCause := E_Heating_RootCause.RC_LOW_SUPPLY_TEMP;
        VO_Confidence := 0.60;
        VO_Error_Score := 0.40;
        VO_Reason_Code := 500;
        VO_Reason_Text := 'Partial cascade capacity';
        RETURN;
    END_IF;
END_IF;

// ======================================================
// LEGACY BOILER / TRANSPORT FALLBACK
// ======================================================
IF NOT L_AnyBoilerOnline THEN
    VO_RootCause := E_Heating_RootCause.RC_BOILER_OFFLINE;
    VO_Confidence := 0.90;
    VO_Error_Score := 0.90;
    VO_Reason_Code := 110;
    VO_Reason_Text := 'No boiler online';
    RETURN;
END_IF;

IF L_AnyBoilerError THEN
    VO_RootCause := E_Heating_RootCause.RC_BOILER_ERROR;
    VO_Confidence := 0.90;
    VO_Error_Score := 0.90;
    VO_Reason_Code := 120;
    VO_Reason_Text := 'Boiler error active';
    RETURN;
END_IF;

IF L_AnyDemand AND NOT L_AnyFlame THEN
    VO_RootCause := E_Heating_RootCause.RC_NO_FLAME;
    VO_Confidence := 0.80;
    VO_Error_Score := 0.80;
    VO_Reason_Code := 130;
    VO_Reason_Text := 'Demand active but no flame';
    RETURN;
END_IF;

// ======================================================
// HYDRAULICS
// ======================================================
IF L_AnyDemand THEN
    IF NOT L_AnyPumpOn THEN
        VO_RootCause := E_Heating_RootCause.RC_PUMP_FAILURE;
        VO_Confidence := 0.80;
        VO_Error_Score := 0.80;
        VO_Reason_Code := 400;
        VO_Reason_Text := 'Demand active but manifold pumps are off';
        RETURN;
    END_IF;

    IF NOT L_AnyValveOpen THEN
        VO_RootCause := E_Heating_RootCause.RC_VALVES_CLOSED;
        VO_Confidence := 0.80;
        VO_Error_Score := 0.80;
        VO_Reason_Code := 410;
        VO_Reason_Text := 'Demand active but manifold valves are closed';
        RETURN;
    END_IF;
END_IF;

// ======================================================
// THERMAL TRANSFER
// ======================================================
IF L_AnyDemand AND L_LowSupply THEN
    VO_RootCause := E_Heating_RootCause.RC_NO_HEAT_TRANSFER;
    VO_Confidence := 0.70;
    VO_Error_Score := 0.70;
    VO_Reason_Code := 420;
    VO_Reason_Text := 'Supply temperature below target under demand';
    RETURN;
END_IF;

// ======================================================
// SENSORS
// ======================================================
IF VI_Sensor_Error THEN
    VO_RootCause := E_Heating_RootCause.RC_SENSOR_ERROR;
    VO_Confidence := 0.70;
    VO_Error_Score := 0.70;
    VO_Reason_Code := 450;
    VO_Reason_Text := 'Heating sensor error active';
    RETURN;
END_IF;

// ======================================================
// NORMAL
// ======================================================
VO_RootCause := E_Heating_RootCause.RC_NONE;
VO_Confidence := 1.0;
VO_Error_Score := 0.0;
VO_Reason_Code := 0;
VO_Reason_Text := 'Heating inference OK';

END_FUNCTION_BLOCK

(* ---- FB_Distributed_Authority_Arbitration.st ---- *)
FUNCTION_BLOCK FB_Distributed_Authority_Arbitration
VAR_INPUT
    VI_Enable : BOOL;
    VI_System_Time_MS : UDINT;
END_VAR
VAR
    L_State : ST_Distributed_Authority_State;
    L_Lease_Expired : BOOL;

    L_Finalized_Runtime_Continuity : BOOL;
END_VAR

IF NOT VI_Enable THEN
    GVL_Distributed_Authority.G_Runtime_Valid := FALSE;
    RETURN;
END_IF;

L_State := (Runtime_Valid := TRUE);
L_State.Runtime_System_Time_MS := VI_System_Time_MS;

L_State.Controller_Id :=
    GVL_Distributed_Runtime.G_Local_Node_State.Controller_Id;

L_State.Runtime_Node_Id :=
    GVL_Distributed_Runtime.G_Local_Node_State.Runtime_Node_Id;

L_State.Authority_Domain_Id :=
    GVL_Distributed_Runtime.G_Local_Node_State.Authority_Domain_Id;

L_State.Authority_Election_Active := TRUE;

L_Lease_Expired :=
    (VI_System_Time_MS - GVL_Distributed_Authority.G_Authority_Lease_Start_MS)
    > GVL_Distributed_Authority.G_Authority_Lease_Duration_MS;

L_State.Authority_Lease_Expired := L_Lease_Expired;
L_State.Authority_Lease_Valid := NOT L_Lease_Expired;

L_State.Replication_Consensus_Healthy :=
    GVL_Distributed_Runtime.G_Distributed_Replication_Healthy;

L_State.Replication_Consensus_Stale :=
    NOT GVL_Distributed_Runtime.G_Distributed_Replication_Healthy;

// Finalized runtime continuity proof chain.
L_Finalized_Runtime_Continuity :=
    GVL_SEMANTIC_PROGRESS.Semantic_Forward_Progress_Valid
    AND GVL_SEMANTIC_PROGRESS.Semantic_Execution_Continuity_OK
    AND NOT GVL_SEMANTIC_PROGRESS.Semantic_Progress_Lease_Expired
    AND NOT GVL_SEMANTIC_PROGRESS.Semantic_Progress_Quarantine_Active
    AND GVL_RUNTIME_SNAPSHOT.Snapshot_Frozen
    AND GVL_RUNTIME_SNAPSHOT.Snapshot_Publication_Allowed
    AND GVL_RUNTIME_SNAPSHOT.Snapshot_Copy_Valid
    AND GVL_RUNTIME_SNAPSHOT.Snapshot_Isolation_Valid
    AND NOT GVL_RUNTIME_SNAPSHOT.Snapshot_Mutation_Detected
    AND GVL_DISTRIBUTED_SNAPSHOT.Distributed_Publication_Reconciled
    AND GVL_DISTRIBUTED_SNAPSHOT.Distributed_Publication_Freeze_Valid
    AND GVL_DISTRIBUTED_SNAPSHOT.Distributed_Snapshot_Consistent
    AND GVL_DISTRIBUTED_COMMIT.Distributed_Commit_Valid
    AND GVL_DISTRIBUTED_COMMIT.Publication_Prepare_Valid
    AND GVL_DISTRIBUTED_COMMIT.Publication_Commit_Confirmed
    AND NOT GVL_DISTRIBUTED_COMMIT.Peer_Commit_Mismatch
    AND NOT GVL_DISTRIBUTED_COMMIT.Commit_Lease_Expired
    AND GVL_OUTPUT_EPOCH.Output_Publication_Valid
    AND GVL_OUTPUT_EPOCH.Output_Runtime_Epoch_Valid
    AND NOT GVL_OUTPUT_EPOCH.Output_Lease_Expired
    AND NOT GVL_OUTPUT_EPOCH.Output_Forced_Safe_Decay
    AND GVL_COMMAND_VERIFY.PreOutput_Barrier_OK
    AND NOT GVL_COMMAND_VERIFY.PreOutput_Block_IO;

// Distributed pre-authority safety barrier.
L_State.Distributed_Safety_Barrier_OK :=
    GVL_Runtime_Restart_Continuity.G_Runtime_Valid
    AND NOT GVL_Config_Activation.G_Config_Quarantine_Active
    AND NOT GVL_Distributed_Runtime.G_Split_Brain_Suspected
    AND GVL_IO_Binding_Runtime.G_Runtime_Valid
    AND L_Finalized_Runtime_Continuity;

IF NOT L_State.Distributed_Safety_Barrier_OK THEN

    L_State.Split_Brain_Blocked := TRUE;
    L_State.Authority_Observer_Only := TRUE;

    L_State.Status_Code := 3;
    L_State.Status_Text :=
        'Distributed authority blocked by safety barrier';

ELSIF L_State.Replication_Consensus_Healthy
   AND NOT L_Lease_Expired
   AND L_Finalized_Runtime_Continuity THEN

    L_State.Authority_Master_Elected := TRUE;

    L_State.Recovery_Authority_Allowed := TRUE;
    L_State.Rollback_Authority_Allowed := TRUE;
    L_State.Quarantine_Authority_Allowed := TRUE;

    L_State.Status_Code := 1;
    L_State.Status_Text :=
        'Distributed master authority active';

ELSE

    L_State.Authority_Backup_Elected := TRUE;

    L_State.Status_Code := 2;
    L_State.Status_Text :=
        'Distributed backup authority active';

END_IF;

GVL_Distributed_Authority.G_Authority_State := L_State;

GVL_Distributed_Authority.G_Split_Brain_Blocked :=
    L_State.Split_Brain_Blocked;

GVL_Distributed_Authority.G_Distributed_Safety_Barrier_OK :=
    L_State.Distributed_Safety_Barrier_OK;

GVL_Distributed_Authority.G_Runtime_Valid := TRUE;
GVL_Distributed_Authority.G_Last_Update_MS := VI_System_Time_MS;
GVL_Distributed_Authority.G_Status_Code := L_State.Status_Code;
GVL_Distributed_Authority.G_Status_Text := L_State.Status_Text;

END_FUNCTION_BLOCK

(* ---- FB_Distributed_Execution_Gates_Runtime.st ---- *)
FUNCTION_BLOCK FB_Distributed_Execution_Gates_Runtime
VAR_INPUT
    VI_Enable : BOOL;
    VI_System_Time_MS : UDINT;
END_VAR
VAR
    L_Allow : BOOL;
    L_Observer_Only : BOOL;
END_VAR

IF NOT VI_Enable THEN
    GVL_Distributed_Execution_Gates.G_Runtime_Valid := FALSE;
    RETURN;
END_IF;

// Observer-only runtime semantics.
// Observer nodes may:
//   - observe runtime state;
//   - receive publications;
//   - participate in diagnostics.
//
// Observer nodes must NEVER:
//   - execute orchestration;
//   - own projections;
//   - execute recovery;
//   - publish physical outputs.
L_Observer_Only :=
    GVL_Distributed_Authority.G_Authority_State.Authority_Observer_Only;

L_Allow :=
    NOT GVL_Cluster_Safety_Barrier.G_Cluster_Execution_Blocked
    AND GVL_Distributed_Authority.G_Authority_State.Authority_Master_Elected
    AND NOT GVL_Distributed_Runtime.G_Split_Brain_Suspected
    AND NOT GVL_Distributed_Projection_Ownership.G_Any_Ownership_Conflict
    AND NOT GVL_Runtime_Sessions.G_Any_Stale_Session
    AND NOT L_Observer_Only;

GVL_Distributed_Execution_Gates.G_Can_Replicate :=
    GVL_Runtime_Bus.G_TX_Healthy
    AND GVL_Runtime_Bus.G_RX_Healthy;

GVL_Distributed_Execution_Gates.G_Can_Execute :=
    L_Allow;

GVL_Distributed_Execution_Gates.G_Can_Orchestrate :=
    L_Allow
    AND GVL_Distributed_Orchestration.G_Distributed_Scheduler_Healthy;

GVL_Distributed_Execution_Gates.G_Can_Recover :=
    L_Allow
    AND NOT GVL_Distributed_Recovery_Lock.G_Recovery_Execution_Blocked;

GVL_Distributed_Execution_Gates.G_Can_Rollback :=
    L_Allow
    AND NOT GVL_Distributed_Recovery_Lock.G_Rollback_Execution_Blocked;

GVL_Distributed_Execution_Gates.G_Can_Own_Projection :=
    L_Allow
    AND NOT GVL_Distributed_Projection_Ownership.G_Any_Projection_Blocked;

GVL_Distributed_Execution_Gates.G_Runtime_Valid := TRUE;
GVL_Distributed_Execution_Gates.G_Last_Update_MS :=
    VI_System_Time_MS;

IF L_Observer_Only THEN

    GVL_Distributed_Execution_Gates.G_Status_Code := 2;
    GVL_Distributed_Execution_Gates.G_Status_Text :=
        'Distributed runtime observer-only';

ELSIF L_Allow THEN

    GVL_Distributed_Execution_Gates.G_Status_Code := 0;
    GVL_Distributed_Execution_Gates.G_Status_Text :=
        'Distributed execution gates open';

ELSE

    GVL_Distributed_Execution_Gates.G_Status_Code := 1;
    GVL_Distributed_Execution_Gates.G_Status_Text :=
        'Distributed execution gates restricted';

END_IF;

END_FUNCTION_BLOCK

(* ---- FB_Distributed_Orchestration_Runtime.st ---- *)
FUNCTION_BLOCK FB_Distributed_Orchestration_Runtime
VAR_INPUT
    VI_Enable : BOOL;
    VI_System_Time_MS : UDINT;
END_VAR
VAR
    L_State : ST_Distributed_Orchestration_State;

    L_Finalized_Runtime_Continuity : BOOL;
END_VAR

IF NOT VI_Enable THEN
    GVL_Distributed_Orchestration.G_Runtime_Valid := FALSE;
    RETURN;
END_IF;

L_State := (Runtime_Valid := TRUE);
L_State.Runtime_System_Time_MS := VI_System_Time_MS;

L_State.Orchestration_Sequence_Id :=
    GVL_Distributed_Orchestration.G_Last_Distributed_Sequence_Id + 1;

L_State.Distributed_Execution_Active := TRUE;

L_State.Cross_Node_Isolation_Required :=
    GVL_Distributed_Orchestration.G_Cross_Node_Isolation_Active;

L_State.Cross_Node_Recovery_Required :=
    GVL_Distributed_Orchestration.G_Cross_Node_Recovery_Active;

L_State.Cross_Node_Rollback_Required :=
    GVL_Distributed_Orchestration.G_Cross_Node_Rollback_Active;

// Finalized runtime continuity proof chain.
L_Finalized_Runtime_Continuity :=
    GVL_SEMANTIC_PROGRESS.Semantic_Forward_Progress_Valid
    AND GVL_SEMANTIC_PROGRESS.Semantic_Execution_Continuity_OK
    AND NOT GVL_SEMANTIC_PROGRESS.Semantic_Progress_Lease_Expired
    AND NOT GVL_SEMANTIC_PROGRESS.Semantic_Progress_Quarantine_Active
    AND GVL_RUNTIME_SNAPSHOT.Snapshot_Frozen
    AND GVL_RUNTIME_SNAPSHOT.Snapshot_Publication_Allowed
    AND GVL_RUNTIME_SNAPSHOT.Snapshot_Copy_Valid
    AND GVL_RUNTIME_SNAPSHOT.Snapshot_Isolation_Valid
    AND NOT GVL_RUNTIME_SNAPSHOT.Snapshot_Mutation_Detected
    AND GVL_DISTRIBUTED_SNAPSHOT.Distributed_Publication_Reconciled
    AND GVL_DISTRIBUTED_SNAPSHOT.Distributed_Publication_Freeze_Valid
    AND GVL_DISTRIBUTED_SNAPSHOT.Distributed_Snapshot_Consistent
    AND GVL_DISTRIBUTED_COMMIT.Distributed_Commit_Valid
    AND GVL_DISTRIBUTED_COMMIT.Publication_Prepare_Valid
    AND GVL_DISTRIBUTED_COMMIT.Publication_Commit_Confirmed
    AND NOT GVL_DISTRIBUTED_COMMIT.Peer_Commit_Mismatch
    AND NOT GVL_DISTRIBUTED_COMMIT.Commit_Lease_Expired
    AND GVL_OUTPUT_EPOCH.Output_Publication_Valid
    AND GVL_OUTPUT_EPOCH.Output_Runtime_Epoch_Valid
    AND NOT GVL_OUTPUT_EPOCH.Output_Lease_Expired
    AND NOT GVL_OUTPUT_EPOCH.Output_Forced_Safe_Decay
    AND GVL_COMMAND_VERIFY.PreOutput_Barrier_OK
    AND NOT GVL_COMMAND_VERIFY.PreOutput_Block_IO;

L_State.Distributed_Scheduler_Healthy :=
    GVL_Runtime_Bus.G_TX_Healthy
    AND GVL_Distributed_Runtime.G_Distributed_Authority_Healthy
    AND L_Finalized_Runtime_Continuity;

L_State.Distributed_Timing_Window_Valid :=
    GVL_Distributed_Authority.G_Distributed_Safety_Barrier_OK
    AND L_Finalized_Runtime_Continuity;

IF L_State.Distributed_Scheduler_Healthy
   AND L_State.Distributed_Timing_Window_Valid THEN

    L_State.Distributed_Projection_Granted := TRUE;
    L_State.Distributed_Recovery_Allowed := TRUE;
    L_State.Distributed_Rollback_Allowed := TRUE;

    L_State.Status_Code := 0;
    L_State.Status_Text :=
        'Distributed orchestration runtime healthy';

ELSE

    L_State.Distributed_Projection_Blocked := TRUE;
    L_State.Distributed_Conflict_Detected := TRUE;

    L_State.Status_Code := 2;
    L_State.Status_Text :=
        'Distributed orchestration blocked';

END_IF;

IF GVL_Distributed_Runtime.G_Split_Brain_Suspected THEN

    L_State.Distributed_Split_Execution_Suspected := TRUE;

    L_State.Distributed_Projection_Blocked := TRUE;

    L_State.Status_Code := 3;
    L_State.Status_Text :=
        'Distributed split execution suspected';

END_IF;

GVL_Distributed_Orchestration.G_Orchestration_State :=
    L_State;

GVL_Distributed_Orchestration.G_Last_Distributed_Sequence_Id :=
    L_State.Orchestration_Sequence_Id;

GVL_Distributed_Orchestration.G_Distributed_Projection_Healthy :=
    L_State.Distributed_Projection_Granted;

GVL_Distributed_Orchestration.G_Distributed_Scheduler_Healthy :=
    L_State.Distributed_Scheduler_Healthy;

GVL_Distributed_Orchestration.G_Runtime_Valid := TRUE;
GVL_Distributed_Orchestration.G_Last_Update_MS := VI_System_Time_MS;
GVL_Distributed_Orchestration.G_Status_Code := L_State.Status_Code;
GVL_Distributed_Orchestration.G_Status_Text := L_State.Status_Text;

END_FUNCTION_BLOCK

(* ---- FB_Distributed_Projection_Ownership_Runtime.st ---- *)
FUNCTION_BLOCK FB_Distributed_Projection_Ownership_Runtime
VAR_INPUT
    VI_Enable : BOOL;
    VI_System_Time_MS : UDINT;
END_VAR
VAR
    L_i : INT;
    L_Ownership : ST_Distributed_Projection_Ownership;

    L_Any_Conflict : BOOL;
    L_Any_Stale : BOOL;
    L_Any_Blocked : BOOL;

    L_Finalized_Runtime_Continuity : BOOL;
END_VAR

IF NOT VI_Enable THEN
    GVL_Distributed_Projection_Ownership.G_Runtime_Valid := FALSE;
    RETURN;
END_IF;

// Finalized runtime continuity proof chain.
L_Finalized_Runtime_Continuity :=
    GVL_SEMANTIC_PROGRESS.Semantic_Forward_Progress_Valid
    AND GVL_SEMANTIC_PROGRESS.Semantic_Execution_Continuity_OK
    AND NOT GVL_SEMANTIC_PROGRESS.Semantic_Progress_Lease_Expired
    AND NOT GVL_SEMANTIC_PROGRESS.Semantic_Progress_Quarantine_Active
    AND GVL_RUNTIME_SNAPSHOT.Snapshot_Frozen
    AND GVL_RUNTIME_SNAPSHOT.Snapshot_Publication_Allowed
    AND GVL_RUNTIME_SNAPSHOT.Snapshot_Copy_Valid
    AND GVL_RUNTIME_SNAPSHOT.Snapshot_Isolation_Valid
    AND NOT GVL_RUNTIME_SNAPSHOT.Snapshot_Mutation_Detected
    AND GVL_DISTRIBUTED_SNAPSHOT.Distributed_Publication_Reconciled
    AND GVL_DISTRIBUTED_SNAPSHOT.Distributed_Publication_Freeze_Valid
    AND GVL_DISTRIBUTED_SNAPSHOT.Distributed_Snapshot_Consistent
    AND GVL_DISTRIBUTED_COMMIT.Distributed_Commit_Valid
    AND GVL_DISTRIBUTED_COMMIT.Publication_Prepare_Valid
    AND GVL_DISTRIBUTED_COMMIT.Publication_Commit_Confirmed
    AND NOT GVL_DISTRIBUTED_COMMIT.Peer_Commit_Mismatch
    AND NOT GVL_DISTRIBUTED_COMMIT.Commit_Lease_Expired
    AND GVL_OUTPUT_EPOCH.Output_Publication_Valid
    AND GVL_OUTPUT_EPOCH.Output_Runtime_Epoch_Valid
    AND NOT GVL_OUTPUT_EPOCH.Output_Lease_Expired
    AND NOT GVL_OUTPUT_EPOCH.Output_Forced_Safe_Decay
    AND GVL_COMMAND_VERIFY.PreOutput_Barrier_OK
    AND NOT GVL_COMMAND_VERIFY.PreOutput_Block_IO;

FOR L_i := 1 TO 128 DO

    L_Ownership :=
        GVL_Distributed_Projection_Ownership.G_Projection_Ownership[L_i];

    IF L_Ownership.Ownership_Valid THEN

        L_Ownership.Runtime_System_Time_MS :=
            VI_System_Time_MS;

        // Ownership becomes stale if runtime sessions unhealthy.
        IF GVL_Runtime_Sessions.G_Any_Stale_Session THEN

            L_Ownership.Ownership_Stale := TRUE;
            L_Any_Stale := TRUE;

        END_IF;

        // Finalized continuity loss invalidates ownership.
        IF NOT L_Finalized_Runtime_Continuity THEN

            L_Ownership.Ownership_Stale := TRUE;
            L_Ownership.Projection_Blocked := TRUE;

            L_Any_Stale := TRUE;
            L_Any_Blocked := TRUE;

        END_IF;

        // Hard conflict prevention.
        IF GVL_Distributed_Runtime.G_Split_Brain_Suspected THEN

            L_Ownership.Ownership_Conflict := TRUE;
            L_Ownership.Projection_Blocked := TRUE;

            L_Any_Conflict := TRUE;
            L_Any_Blocked := TRUE;

        END_IF;

        // Distributed execution authority.
        IF GVL_Distributed_Authority.G_Authority_State.Authority_Master_Elected
           AND NOT L_Ownership.Ownership_Conflict
           AND NOT L_Ownership.Ownership_Stale
           AND L_Finalized_Runtime_Continuity THEN

            L_Ownership.Ownership_Granted := TRUE;
            L_Ownership.Distributed_Execution_Allowed := TRUE;
            L_Ownership.Distributed_Recovery_Allowed := TRUE;

            L_Ownership.Status_Code := 0;
            L_Ownership.Status_Text :=
                'Distributed projection ownership granted';

        ELSE

            L_Ownership.Ownership_Revoked := TRUE;
            L_Ownership.Projection_Blocked := TRUE;

            L_Any_Blocked := TRUE;

            L_Ownership.Status_Code := 2;
            L_Ownership.Status_Text :=
                'Distributed projection ownership blocked';

        END_IF;

        GVL_Distributed_Projection_Ownership.G_Projection_Ownership[L_i] :=
            L_Ownership;

    END_IF;

END_FOR;

GVL_Distributed_Projection_Ownership.G_Any_Ownership_Conflict :=
    L_Any_Conflict;

GVL_Distributed_Projection_Ownership.G_Any_Ownership_Stale :=
    L_Any_Stale;

GVL_Distributed_Projection_Ownership.G_Any_Projection_Blocked :=
    L_Any_Blocked;

GVL_Distributed_Projection_Ownership.G_Runtime_Valid := TRUE;
GVL_Distributed_Projection_Ownership.G_Last_Update_MS :=
    VI_System_Time_MS;

IF L_Any_Conflict THEN
    GVL_Distributed_Projection_Ownership.G_Status_Code := 3;
    GVL_Distributed_Projection_Ownership.G_Status_Text :=
        'Distributed projection ownership conflict detected';
ELSIF L_Any_Stale THEN
    GVL_Distributed_Projection_Ownership.G_Status_Code := 2;
    GVL_Distributed_Projection_Ownership.G_Status_Text :=
        'Distributed projection ownership stale';
ELSIF L_Any_Blocked THEN
    GVL_Distributed_Projection_Ownership.G_Status_Code := 1;
    GVL_Distributed_Projection_Ownership.G_Status_Text :=
        'Distributed projection ownership blocked';
ELSE
    GVL_Distributed_Projection_Ownership.G_Status_Code := 0;
    GVL_Distributed_Projection_Ownership.G_Status_Text :=
        'Distributed projection ownership healthy';
END_IF;

END_FUNCTION_BLOCK

(* ---- FB_Distributed_Recovery_Lock_Runtime.st ---- *)
FUNCTION_BLOCK FB_Distributed_Recovery_Lock_Runtime
VAR_INPUT
    VI_Enable : BOOL;
    VI_System_Time_MS : UDINT;
END_VAR
VAR
    L_Lock : ST_Distributed_Recovery_Lock;
END_VAR

IF NOT VI_Enable THEN
    GVL_Distributed_Recovery_Lock.G_Runtime_Valid := FALSE;
    RETURN;
END_IF;

L_Lock := GVL_Distributed_Recovery_Lock.G_Recovery_Lock;

L_Lock.Runtime_System_Time_MS := VI_System_Time_MS;
L_Lock.Lock_Valid := TRUE;

// Cluster-exclusive recovery execution lock.
IF GVL_Distributed_Runtime.G_Split_Brain_Suspected
   OR GVL_Distributed_Projection_Ownership.G_Any_Ownership_Conflict
   OR GVL_Runtime_Sessions.G_Any_Stale_Session THEN

    L_Lock.Lock_Conflict := TRUE;
    L_Lock.Distributed_Execution_Allowed := FALSE;

    GVL_Distributed_Recovery_Lock.G_Recovery_Execution_Blocked := TRUE;
    GVL_Distributed_Recovery_Lock.G_Rollback_Execution_Blocked := TRUE;
    GVL_Distributed_Recovery_Lock.G_Reopen_Execution_Blocked := TRUE;

    L_Lock.Status_Code := 3;
    L_Lock.Status_Text :=
        'Distributed recovery execution locked';

ELSE

    L_Lock.Recovery_Lock_Active := TRUE;
    L_Lock.Distributed_Execution_Allowed := TRUE;

    GVL_Distributed_Recovery_Lock.G_Recovery_Execution_Blocked := FALSE;
    GVL_Distributed_Recovery_Lock.G_Rollback_Execution_Blocked := FALSE;
    GVL_Distributed_Recovery_Lock.G_Reopen_Execution_Blocked := FALSE;

    L_Lock.Status_Code := 0;
    L_Lock.Status_Text :=
        'Distributed recovery lock healthy';

END_IF;

GVL_Distributed_Recovery_Lock.G_Recovery_Lock := L_Lock;

GVL_Distributed_Recovery_Lock.G_Runtime_Valid := TRUE;
GVL_Distributed_Recovery_Lock.G_Last_Update_MS :=
    VI_System_Time_MS;

GVL_Distributed_Recovery_Lock.G_Status_Code :=
    L_Lock.Status_Code;

GVL_Distributed_Recovery_Lock.G_Status_Text :=
    L_Lock.Status_Text;

END_FUNCTION_BLOCK

(* ---- FB_Distributed_Runtime_Continuity.st ---- *)
FUNCTION_BLOCK FB_Distributed_Runtime_Continuity
VAR_INPUT
    VI_Enable : BOOL;
    VI_System_Time_MS : UDINT;
END_VAR
VAR
    L_i : INT;
    L_Node : ST_Distributed_Runtime_Node_State;

    L_Any_Offline : BOOL;
    L_Any_Degraded : BOOL;
    L_Split_Brain : BOOL;
END_VAR

IF NOT VI_Enable THEN
    GVL_Distributed_Runtime.G_Runtime_Valid := FALSE;
    RETURN;
END_IF;

// Local node authoritative runtime state.
GVL_Distributed_Runtime.G_Local_Node_State.Runtime_Valid := TRUE;
GVL_Distributed_Runtime.G_Local_Node_State.Runtime_System_Time_MS :=
    VI_System_Time_MS;

GVL_Distributed_Runtime.G_Local_Node_State.Node_Online := TRUE;

GVL_Distributed_Runtime.G_Local_Node_State.Restart_Continuity_Valid :=
    GVL_Runtime_Restart_Continuity.G_Runtime_Valid;

GVL_Distributed_Runtime.G_Local_Node_State.Quarantine_State_Replicated :=
    NOT GVL_Config_Activation.G_Config_Quarantine_Active;

GVL_Distributed_Runtime.G_Local_Node_State.Recovery_State_Replicated :=
    GVL_Water_Recovery_Runtime.G_Runtime_Valid;

GVL_Distributed_Runtime.G_Local_Node_State.Authority_Allowed :=
    NOT GVL_COMMAND_VERIFY.PreOutput_Block_IO;

GVL_Distributed_Runtime.G_Local_Node_State.Replication_Healthy := TRUE;

FOR L_i := 1 TO 8 DO

    L_Node := GVL_Distributed_Runtime.G_Remote_Node_State[L_i];

    IF L_Node.Runtime_Valid THEN

        IF NOT L_Node.Node_Online THEN
            L_Any_Offline := TRUE;
        END_IF;

        IF L_Node.Node_Degraded
           OR L_Node.Node_Quarantined THEN

            L_Any_Degraded := TRUE;

        END_IF;

        IF L_Node.Authority_Master
           AND GVL_Distributed_Runtime.G_Local_Node_State.Authority_Master THEN

            L_Split_Brain := TRUE;

        END_IF;

    END_IF;

END_FOR;

GVL_Distributed_Runtime.G_Any_Remote_Node_Offline :=
    L_Any_Offline;

GVL_Distributed_Runtime.G_Any_Remote_Node_Degraded :=
    L_Any_Degraded;

GVL_Distributed_Runtime.G_Split_Brain_Suspected :=
    L_Split_Brain;

GVL_Distributed_Runtime.G_Distributed_Replication_Healthy :=
    NOT L_Any_Offline;

GVL_Distributed_Runtime.G_Distributed_Authority_Healthy :=
    NOT L_Split_Brain;

GVL_Distributed_Runtime.G_Runtime_Valid := TRUE;
GVL_Distributed_Runtime.G_Last_Update_MS := VI_System_Time_MS;

IF L_Split_Brain THEN
    GVL_Distributed_Runtime.G_Status_Code := 3;
    GVL_Distributed_Runtime.G_Status_Text :=
        'Distributed split-brain suspected';
ELSIF L_Any_Degraded THEN
    GVL_Distributed_Runtime.G_Status_Code := 2;
    GVL_Distributed_Runtime.G_Status_Text :=
        'Distributed degraded node detected';
ELSIF L_Any_Offline THEN
    GVL_Distributed_Runtime.G_Status_Code := 1;
    GVL_Distributed_Runtime.G_Status_Text :=
        'Distributed offline node detected';
ELSE
    GVL_Distributed_Runtime.G_Status_Code := 0;
    GVL_Distributed_Runtime.G_Status_Text :=
        'Distributed runtime continuity healthy';
END_IF;

END_FUNCTION_BLOCK

(* ---- FB_DryRun_Assertion_Map.st ---- *)
FUNCTION_BLOCK FB_DryRun_Assertion_Map
VAR_INPUT
    VI_Test_Step : INT;
END_VAR

VAR_OUTPUT
    VO_Expected_Result : STRING(220);
END_VAR

CASE VI_Test_Step OF
    1:
        VO_Expected_Result := 'EXPECT: Flood alarm active, leak safety path active, water confirm blocked';
    2:
        VO_Expected_Result := 'EXPECT: Gas alarm active, gas valve close path, gas safety latched';
    3:
        VO_Expected_Result := 'EXPECT: Fire alarm active, smoke safety path, safe-stop tendency';
    4:
        VO_Expected_Result := 'EXPECT: Scenario NONE clamp under SAFE_STOP/FREEZE rules';
    5:
        VO_Expected_Result := 'EXPECT: Scenario forced to AWAY by security policy';
    6:
        VO_Expected_Result := 'EXPECT: Guard denies AWAY->PARTY, scenario remains unchanged';
    7:
        VO_Expected_Result := 'EXPECT: Watchdog root cause and event 11/12 path';
    ELSE
        VO_Expected_Result := 'EXPECT: No active dry-run case';
END_CASE;

// >>> BULK_SYNC_ANCHOR: FB_DryRun_Assertion_Map <<<

(* ---- FB_DryRun_Simulation_Harness.st ---- *)
FUNCTION_BLOCK FB_DryRun_Simulation_Harness
VAR_INPUT
    VI_Enable : BOOL;
    VI_System_Time_MS : UDINT;
END_VAR

VAR_OUTPUT
    VO_Test_Step : INT;
    VO_Status_Msg : STRING(120);
    VO_Inject_Flood : BOOL;
    VO_Inject_Gas : BOOL;
    VO_Inject_Fire : BOOL;
    VO_Inject_SafeStop : BOOL;
    VO_Inject_SecurityArmed : BOOL;
    VO_Request_AwayToParty : BOOL;
    VO_Inject_Watchdog : BOOL;
END_VAR

VAR
    L_Last_Step_Time : UDINT;
END_VAR

IF NOT VI_Enable THEN
    VO_Test_Step := 0;
    VO_Status_Msg := 'Dry run disabled';
    VO_Inject_Flood := FALSE;
    VO_Inject_Gas := FALSE;
    VO_Inject_Fire := FALSE;
    VO_Inject_SafeStop := FALSE;
    VO_Inject_SecurityArmed := FALSE;
    VO_Request_AwayToParty := FALSE;
    VO_Inject_Watchdog := FALSE;
    RETURN;
END_IF;

// reset one-shot style outputs before step dispatch
VO_Inject_Flood := FALSE;
VO_Inject_Gas := FALSE;
VO_Inject_Fire := FALSE;
VO_Inject_SafeStop := FALSE;
VO_Inject_SecurityArmed := FALSE;
VO_Request_AwayToParty := FALSE;
VO_Inject_Watchdog := FALSE;

IF (VI_System_Time_MS - L_Last_Step_Time) < 5000 THEN
    RETURN;
END_IF;

L_Last_Step_Time := VI_System_Time_MS;
VO_Test_Step := VO_Test_Step + 1;

CASE VO_Test_Step OF
    1:
        VO_Inject_Flood := TRUE;
        VO_Status_Msg := 'Dry run: flood case';
    2:
        VO_Inject_Gas := TRUE;
        VO_Status_Msg := 'Dry run: gas case';
    3:
        VO_Inject_Fire := TRUE;
        VO_Status_Msg := 'Dry run: fire case';
    4:
        VO_Inject_SafeStop := TRUE;
        VO_Status_Msg := 'Dry run: safe-stop clamp';
    5:
        VO_Inject_SecurityArmed := TRUE;
        VO_Status_Msg := 'Dry run: policy away';
    6:
        VO_Request_AwayToParty := TRUE;
        VO_Status_Msg := 'Dry run: scenario guard deny';
    7:
        VO_Inject_Watchdog := TRUE;
        VO_Status_Msg := 'Dry run: watchdog case';
    ELSE
        VO_Test_Step := 0;
        VO_Status_Msg := 'Dry run: cycle restart';
END_CASE;

// >>> BULK_SYNC_ANCHOR: FB_DryRun_Simulation_Harness <<<

(* ---- FB_FloorHeating_Controller.st ---- *)
FUNCTION_BLOCK FB_FloorHeating_Controller
VAR_INPUT
    VI_Current_Temp : REAL;
    VI_Config : ST_FloorHeating_Circuit_Config;
    VI_Tariff : ST_Tariff_Config;
    VI_Current_Hour : UINT;
    VI_IsActivePLC : BOOL;
    VI_System_Time_MS : UDINT;
END_VAR
VAR_OUTPUT
    VO_Pump_Run : BOOL;
    VO_Valve_Pos : REAL; // 0..100%
    VO_Valve_Bool : BOOL; // ШИМ выход для термоэлектрического привода
    VO_Effective_Setpoint : REAL;
END_VAR
VAR
    L_Is_Night : BOOL;
    L_PID : FB_PID_Controller;
    L_Last_Time : UDINT;
    L_Cycle_Time_S : REAL;
    L_PWM_Period_MS : UDINT;
    L_PWM_Duty_MS : UDINT;
    L_Current_Phase_MS : UDINT;
    L_PWM_Start_Time : UDINT;
END_VAR

// Вычисление времени цикла
IF L_Last_Time = 0 THEN
    L_Last_Time := VI_System_Time_MS;
    L_Cycle_Time_S := 1.0;
ELSE
    L_Cycle_Time_S := UDINT_TO_REAL((SEL(VI_System_Time_MS >= L_Last_Time, VI_System_Time_MS - L_Last_Time, (4294967295 - L_Last_Time) + VI_System_Time_MS + 1))) / 1000.0;
    L_Last_Time := VI_System_Time_MS;
END_IF;
IF L_Cycle_Time_S <= 0.0 THEN L_Cycle_Time_S := 0.01; END_IF;

// 1. Определение активного тарифа
IF VI_Tariff.Enabled THEN
    IF VI_Tariff.Night_Start_Hour > VI_Tariff.Night_End_Hour THEN
        // Переход через полночь (например, 23:00 - 07:00)
        L_Is_Night := (VI_Current_Hour >= VI_Tariff.Night_Start_Hour) OR (VI_Current_Hour < VI_Tariff.Night_End_Hour);
    ELSE
        // В пределах одного дня
        L_Is_Night := (VI_Current_Hour >= VI_Tariff.Night_Start_Hour) AND (VI_Current_Hour < VI_Tariff.Night_End_Hour);
    END_IF;
ELSE
    L_Is_Night := FALSE;
END_IF;

// 2. Расчет эффективной уставки
VO_Effective_Setpoint := VI_Config.design_temp;
IF L_Is_Night THEN
    VO_Effective_Setpoint := VO_Effective_Setpoint + VI_Tariff.Boost_Delta;
END_IF;

// 3. ПИД-регулирование
L_PID(
    VI_SetPoint := VO_Effective_Setpoint,
    VI_ProcessValue := VI_Current_Temp,
    VI_Kp := VI_Config.pid_kp,
    VI_Tn := 300.0,
    VI_Tv := 0.0,
    VI_Y_Min := 0.0,
    VI_Y_Max := 100.0,
    VI_Cycle_Time_S := L_Cycle_Time_S,
    VO_Output => VO_Valve_Pos
);

// 4. ШИМ-модуляция для термоэлектрического привода
IF VI_Config.pwm_period_s > 0 THEN
    L_PWM_Period_MS := TO_UDINT(VI_Config.pwm_period_s) * 1000;
ELSE
    L_PWM_Period_MS := 600000; // 10 минут
END_IF;

L_Current_Phase_MS := (SEL(VI_System_Time_MS >= L_PWM_Start_Time, VI_System_Time_MS - L_PWM_Start_Time, (4294967295 - L_PWM_Start_Time) + VI_System_Time_MS + 1));
IF L_Current_Phase_MS >= L_PWM_Period_MS THEN
    L_PWM_Start_Time := VI_System_Time_MS - (L_Current_Phase_MS - L_PWM_Period_MS); // Сохраняем остаток для точности
    L_Current_Phase_MS := (SEL(VI_System_Time_MS >= L_PWM_Start_Time, VI_System_Time_MS - L_PWM_Start_Time, (4294967295 - L_PWM_Start_Time) + VI_System_Time_MS + 1));
END_IF;

L_PWM_Duty_MS := TO_UDINT((VO_Valve_Pos / 100.0) * TO_REAL(L_PWM_Period_MS));

IF VI_IsActivePLC THEN
    VO_Pump_Run := (VO_Valve_Pos > 5.0);

    IF VO_Valve_Pos >= 100.0 THEN
        VO_Valve_Bool := TRUE;
    ELSIF VO_Valve_Pos <= 0.0 THEN
        VO_Valve_Bool := FALSE;
    ELSE
        VO_Valve_Bool := (L_Current_Phase_MS <= L_PWM_Duty_MS);
    END_IF;
ELSE
    VO_Pump_Run := FALSE;
    VO_Valve_Bool := FALSE;
END_IF;

(* ---- FB_Forensic_Journal_Runtime.st ---- *)
FUNCTION_BLOCK FB_Forensic_Journal_Runtime
VAR_INPUT
    VI_Enable : BOOL;
    VI_System_Time_MS : UDINT;
END_VAR
VAR
    L_Record : ST_Forensic_Journal_Record;
    L_Write_Index : UINT;
END_VAR

IF NOT VI_Enable THEN
    GVL_Forensic_Journal.G_Runtime_Valid := FALSE;
    RETURN;
END_IF;

L_Write_Index := GVL_Forensic_Journal.G_Write_Index + 1;

IF L_Write_Index > 256 THEN
    L_Write_Index := 1;
END_IF;

IF GVL_Config_Activation.G_Activation_State.Activation_Allowed
   OR GVL_Config_Activation.G_Activation_State.Rollback_Active THEN

    L_Record.Record_Valid := TRUE;
    L_Record.Event_Time_MS := VI_System_Time_MS;
    L_Record.Event_Id := GVL_Forensic_Journal.G_Last_Event_Id + 1;

    L_Record.Config_Version := GVL_Config_Activation.G_Activation_State.Active_Version;
    L_Record.Topology_Version := GVL_Water_Topology_Config.G_Active_Config_Version;

    IF GVL_Config_Activation.G_Activation_State.Rollback_Active THEN
        L_Record.Rollback_Event := TRUE;
        L_Record.Event_Class := 2;
        L_Record.Event_Severity := 2;
        L_Record.Event_Text := 'Topology rollback activated';
        GVL_Forensic_Journal.G_Last_Rollback_Event_Id := L_Record.Event_Id;
    ELSE
        L_Record.Activation_Event := TRUE;
        L_Record.Event_Class := 1;
        L_Record.Event_Severity := 1;
        L_Record.Event_Text := 'Topology activation completed';
        GVL_Forensic_Journal.G_Last_Activation_Event_Id := L_Record.Event_Id;
    END_IF;

    GVL_Forensic_Journal.G_Journal[L_Write_Index] := L_Record;
    GVL_Forensic_Journal.G_Last_Event_Id := L_Record.Event_Id;
    GVL_Forensic_Journal.G_Write_Index := L_Write_Index;
END_IF;

IF GVL_Runtime_Restart_Continuity.G_Continuity_State.Restore_Completed THEN
    L_Write_Index := GVL_Forensic_Journal.G_Write_Index + 1;

    IF L_Write_Index > 256 THEN
        L_Write_Index := 1;
    END_IF;

    L_Record.Record_Valid := TRUE;
    L_Record.Event_Time_MS := VI_System_Time_MS;
    L_Record.Event_Id := GVL_Forensic_Journal.G_Last_Event_Id + 1;
    L_Record.Restart_Event := TRUE;
    L_Record.Event_Class := 3;
    L_Record.Event_Severity := 1;
    L_Record.Config_Version := GVL_Runtime_Restart_Continuity.G_Continuity_State.Active_Config_Version;
    L_Record.Event_Text := 'Warm restart continuity restored';

    GVL_Forensic_Journal.G_Journal[L_Write_Index] := L_Record;
    GVL_Forensic_Journal.G_Last_Event_Id := L_Record.Event_Id;
    GVL_Forensic_Journal.G_Write_Index := L_Write_Index;
    GVL_Forensic_Journal.G_Last_Restart_Event_Id := L_Record.Event_Id;
END_IF;

IF GVL_Config_Activation.G_Config_Quarantine_Active THEN
    L_Write_Index := GVL_Forensic_Journal.G_Write_Index + 1;

    IF L_Write_Index > 256 THEN
        L_Write_Index := 1;
    END_IF;

    L_Record.Record_Valid := TRUE;
    L_Record.Event_Time_MS := VI_System_Time_MS;
    L_Record.Event_Id := GVL_Forensic_Journal.G_Last_Event_Id + 1;
    L_Record.Quarantine_Event := TRUE;
    L_Record.Event_Class := 4;
    L_Record.Event_Severity := 3;
    L_Record.Config_Version := GVL_Config_Activation.G_Activation_State.Staged_Version;
    L_Record.Event_Text := 'Config quarantine active';

    GVL_Forensic_Journal.G_Journal[L_Write_Index] := L_Record;
    GVL_Forensic_Journal.G_Last_Event_Id := L_Record.Event_Id;
    GVL_Forensic_Journal.G_Write_Index := L_Write_Index;
END_IF;

GVL_Forensic_Journal.G_Runtime_Valid := TRUE;
GVL_Forensic_Journal.G_Last_Update_MS := VI_System_Time_MS;
GVL_Forensic_Journal.G_Status_Code := 0;
GVL_Forensic_Journal.G_Status_Text := 'Persistent forensic journal active';

END_FUNCTION_BLOCK

(* ---- FB_Gas_Smoke_Manager.st ---- *)
FUNCTION_BLOCK FB_Gas_Smoke_Manager
VAR_INPUT
    VI_System_Time_MS : UDINT;
    VI_IsActivePLC    : BOOL;
    VI_Mute_Request   : BOOL;
END_VAR

VAR_IN_OUT
    VI_Methane_LEL    : ARRAY[1..GVL_CONSTANTS.C_MAX_METHANE_SENSORS] OF REAL;
    VI_CO_PPM         : ARRAY[1..GVL_CONSTANTS.C_MAX_CO_SENSORS] OF REAL;
    VI_Smoke_Sensors  : ARRAY[1..GVL_CONSTANTS.C_MAX_SMOKE_SENSORS] OF BOOL;
END_VAR

VAR_OUTPUT
    // Health signals
    VO_Smoke_Detected           : BOOL;
    VO_Gas_Detected             : BOOL; // Compatible methane alarm/critical summary.
    VO_Methane_Warning_Level    : BOOL;
    VO_Methane_Alarm_Level      : BOOL;
    VO_Methane_Critical_Level   : BOOL;
    VO_CO_Warning_Level         : BOOL;
    VO_CO_Alarm_Level           : BOOL;
    VO_Status_Msg               : STRING(200);
END_VAR

VAR
    L_Methane_Max   : REAL;
    L_CO_Max        : REAL;
    L_CO_Max_Index  : INT;
    L_Smoke_Count   : UINT;
    L_Smoke_Active  : BOOL;
    L_i             : INT;
    L_Group         : INT;
    L_A             : INT;
    L_B             : INT;

    L_CO_Timer_30ppm  : FB_System_Timer;
    L_CO_Timer_70ppm  : FB_System_Timer;
    L_CO_Timer_400ppm : FB_System_Timer;

    L_CO_Level_30   : BOOL;
    L_CO_Level_70   : BOOL;
    L_CO_Level_400  : BOOL;

    L_Smoke_Timer : ARRAY[1..GVL_CONSTANTS.C_MAX_SMOKE_SENSORS] OF FB_System_Timer;
END_VAR

IF NOT VI_IsActivePLC THEN RETURN; END_IF;

// Reset outputs
VO_Smoke_Detected := FALSE;
VO_Gas_Detected := FALSE;
VO_Methane_Warning_Level := FALSE;
VO_Methane_Alarm_Level := FALSE;
VO_Methane_Critical_Level := FALSE;
VO_CO_Warning_Level := FALSE;
VO_CO_Alarm_Level := FALSE;
VO_Status_Msg := 'ОК';

// --- Methane ---
L_Methane_Max := 0.0;
FOR L_i := 1 TO GVL_CONSTANTS.C_MAX_METHANE_SENSORS DO
    IF VI_Methane_LEL[L_i] > L_Methane_Max THEN
        L_Methane_Max := VI_Methane_LEL[L_i];
    END_IF;
END_FOR;

VO_Methane_Warning_Level := (L_Methane_Max >= 10.0);
VO_Methane_Alarm_Level := (L_Methane_Max >= 20.0);
VO_Methane_Critical_Level := (L_Methane_Max >= 40.0);
VO_Gas_Detected := VO_Methane_Alarm_Level OR VO_Methane_Critical_Level;

// --- CO ---
L_CO_Max := 0.0;
L_CO_Max_Index := 0;
FOR L_i := 1 TO GVL_CONSTANTS.C_MAX_CO_SENSORS DO
    IF VI_CO_PPM[L_i] > L_CO_Max THEN
        L_CO_Max := VI_CO_PPM[L_i];
        L_CO_Max_Index := L_i;
    END_IF;
END_FOR;

L_CO_Level_30 := (L_CO_Max >= 30.0);
L_CO_Level_70 := (L_CO_Max >= 70.0);
L_CO_Level_400 := (L_CO_Max >= 400.0);

L_CO_Timer_30ppm(IN := L_CO_Level_30, PT := T#8h, VI_System_Time_MS := VI_System_Time_MS);
L_CO_Timer_70ppm(IN := L_CO_Level_70, PT := T#1h, VI_System_Time_MS := VI_System_Time_MS);
L_CO_Timer_400ppm(IN := L_CO_Level_400, PT := T#15m, VI_System_Time_MS := VI_System_Time_MS);

IF L_CO_Timer_30ppm.Q THEN
    VO_CO_Warning_Level := TRUE;
END_IF;

IF L_CO_Timer_70ppm.Q OR L_CO_Timer_400ppm.Q THEN
    VO_CO_Alarm_Level := TRUE;
END_IF;

GVL_CO_EXPOSURE.G_CO_Max_PPM := L_CO_Max;
GVL_CO_EXPOSURE.G_CO_Max_Sensor_Index := L_CO_Max_Index;
GVL_CO_EXPOSURE.G_Level_30ppm_Active := L_CO_Level_30;
GVL_CO_EXPOSURE.G_Level_70ppm_Active := L_CO_Level_70;
GVL_CO_EXPOSURE.G_Level_400ppm_Active := L_CO_Level_400;
GVL_CO_EXPOSURE.G_Timer_30ppm_ET := L_CO_Timer_30ppm.ET;
GVL_CO_EXPOSURE.G_Timer_70ppm_ET := L_CO_Timer_70ppm.ET;
GVL_CO_EXPOSURE.G_Timer_400ppm_ET := L_CO_Timer_400ppm.ET;
GVL_CO_EXPOSURE.G_Timer_30ppm_Q := L_CO_Timer_30ppm.Q;
GVL_CO_EXPOSURE.G_Timer_70ppm_Q := L_CO_Timer_70ppm.Q;
GVL_CO_EXPOSURE.G_Timer_400ppm_Q := L_CO_Timer_400ppm.Q;
GVL_CO_EXPOSURE.G_Warning_Active := VO_CO_Warning_Level;
GVL_CO_EXPOSURE.G_Alarm_Active := VO_CO_Alarm_Level;
GVL_CO_EXPOSURE.G_Last_Update_MS := VI_System_Time_MS;

IF VO_CO_Alarm_Level THEN
    GVL_CO_EXPOSURE.G_Status_Text := 'CO alarm exposure threshold reached';
ELSIF VO_CO_Warning_Level THEN
    GVL_CO_EXPOSURE.G_Status_Text := 'CO warning exposure threshold reached';
ELSIF L_CO_Level_400 THEN
    GVL_CO_EXPOSURE.G_Status_Text := 'CO 400ppm exposure accumulating';
ELSIF L_CO_Level_70 THEN
    GVL_CO_EXPOSURE.G_Status_Text := 'CO 70ppm exposure accumulating';
ELSIF L_CO_Level_30 THEN
    GVL_CO_EXPOSURE.G_Status_Text := 'CO 30ppm exposure accumulating';
ELSE
    GVL_CO_EXPOSURE.G_Status_Text := 'CO exposure idle';
END_IF;

// --- Smoke ---
L_Smoke_Count := 0;
L_Smoke_Active := FALSE;
GVL_SMOKE_VERIFICATION.G_Verified_By_Pair := FALSE;
GVL_SMOKE_VERIFICATION.G_Verified_By_Timer := FALSE;
GVL_SMOKE_VERIFICATION.G_Verified_Group := 0;
GVL_SMOKE_VERIFICATION.G_Any_Smoke_Input_Active := FALSE;

FOR L_i := 1 TO 3 DO
    GVL_SMOKE_VERIFICATION.G_Group_Active[L_i] := FALSE;
    GVL_SMOKE_VERIFICATION.G_Group_Pair_Confirmed[L_i] := FALSE;
    GVL_SMOKE_VERIFICATION.G_Group_Timer_Confirmed[L_i] := FALSE;
END_FOR;

FOR L_i := 1 TO GVL_CONSTANTS.C_MAX_SMOKE_SENSORS DO
    L_Smoke_Timer[L_i](IN := VI_Smoke_Sensors[L_i], PT := T#30s, VI_System_Time_MS := VI_System_Time_MS);

    IF VI_Smoke_Sensors[L_i] THEN
        L_Smoke_Count := L_Smoke_Count + 1;
        GVL_SMOKE_VERIFICATION.G_Any_Smoke_Input_Active := TRUE;
    END_IF;
END_FOR;

FOR L_Group := 1 TO 3 DO
    L_A := (L_Group * 2) - 1;
    L_B := L_Group * 2;

    IF (L_A <= GVL_CONSTANTS.C_MAX_SMOKE_SENSORS) AND (L_B <= GVL_CONSTANTS.C_MAX_SMOKE_SENSORS) THEN
        GVL_SMOKE_VERIFICATION.G_Group_Active[L_Group] :=
            VI_Smoke_Sensors[L_A] OR VI_Smoke_Sensors[L_B];

        GVL_SMOKE_VERIFICATION.G_Group_Pair_Confirmed[L_Group] :=
            VI_Smoke_Sensors[L_A] AND VI_Smoke_Sensors[L_B];

        GVL_SMOKE_VERIFICATION.G_Group_Timer_Confirmed[L_Group] :=
            L_Smoke_Timer[L_A].Q OR L_Smoke_Timer[L_B].Q;

        IF GVL_SMOKE_VERIFICATION.G_Group_Pair_Confirmed[L_Group] OR
           GVL_SMOKE_VERIFICATION.G_Group_Timer_Confirmed[L_Group] THEN
            L_Smoke_Active := TRUE;

            IF GVL_SMOKE_VERIFICATION.G_Verified_Group = 0 THEN
                GVL_SMOKE_VERIFICATION.G_Verified_Group := L_Group;
            END_IF;

            IF GVL_SMOKE_VERIFICATION.G_Group_Pair_Confirmed[L_Group] THEN
                GVL_SMOKE_VERIFICATION.G_Verified_By_Pair := TRUE;
            END_IF;

            IF GVL_SMOKE_VERIFICATION.G_Group_Timer_Confirmed[L_Group] THEN
                GVL_SMOKE_VERIFICATION.G_Verified_By_Timer := TRUE;
            END_IF;
        END_IF;
    END_IF;
END_FOR;

GVL_SMOKE_VERIFICATION.G_Smoke_Active_Count := L_Smoke_Count;
GVL_SMOKE_VERIFICATION.G_Verified := L_Smoke_Active;
GVL_SMOKE_VERIFICATION.G_Last_Update_MS := VI_System_Time_MS;

IF L_Smoke_Active THEN
    VO_Smoke_Detected := TRUE;
    CASE GVL_SMOKE_VERIFICATION.G_Verified_Group OF
        1:
            GVL_SMOKE_VERIFICATION.G_Status_Text := 'Smoke verified: basement group';
        2:
            GVL_SMOKE_VERIFICATION.G_Status_Text := 'Smoke verified: floor 1 group';
        3:
            GVL_SMOKE_VERIFICATION.G_Status_Text := 'Smoke verified: floor 2 group';
    ELSE
            GVL_SMOKE_VERIFICATION.G_Status_Text := 'Smoke verified';
    END_CASE;
ELSE
    IF GVL_SMOKE_VERIFICATION.G_Any_Smoke_Input_Active THEN
        GVL_SMOKE_VERIFICATION.G_Status_Text := 'Smoke input active - waiting verification';
    ELSE
        GVL_SMOKE_VERIFICATION.G_Status_Text := 'Smoke verification idle';
    END_IF;
END_IF;

// Status
IF VO_Smoke_Detected THEN
    VO_Status_Msg := 'ПОЖАР';
ELSIF VO_Methane_Critical_Level THEN
    VO_Status_Msg := 'КРИТИЧЕСКИЙ МЕТАН';
ELSIF VO_Methane_Alarm_Level THEN
    VO_Status_Msg := 'УТЕЧКА ГАЗА';
ELSIF VO_Methane_Warning_Level THEN
    VO_Status_Msg := 'ПРЕДУПРЕЖДЕНИЕ МЕТАН';
ELSIF VO_CO_Alarm_Level THEN
    VO_Status_Msg := 'КРИТИЧЕСКИЙ CO';
ELSIF VO_CO_Warning_Level THEN
    VO_Status_Msg := 'ПОВЫШЕННЫЙ CO';
ELSE
    VO_Status_Msg := 'ОК';
END_IF;
// >>> BULK_SYNC_ANCHOR: FB_Gas_Smoke_Manager <<<
END_FUNCTION_BLOCK

(* ---- FB_Gateway_Interface.st ---- *)
FUNCTION_BLOCK FB_Gateway_Interface
VAR_INPUT
    VI_System_Time_MS           : UDINT;
    VI_Local_PLC_Role           : E_PLC_ROLE;
    VI_Incoming_Command         : ST_Gateway_Command;
    VI_Command_Received         : BOOL;

    VI_Outdoor_Temp             : REAL;
    VI_Security_Armed           : BOOL;
    VI_Flood_Alarm_Active       : BOOL;
    VI_Gas_Alarm_Active         : BOOL;
    VI_Fire_Alarm_Active        : BOOL;
    VI_Methane_Concentration    : REAL;
    VI_Active_Scenario          : E_SCENARIO_TYPE;

    VI_Send_2FA_Req             : BOOL;
    VI_2FA_Code                 : STRING(6);
END_VAR

VAR_IN_OUT
    VI_FloorHeating_Temps       : ARRAY[1..GVL_CONSTANTS.C_MAX_HEATING_CIRCUITS] OF REAL;
    VI_Room_Temps               : ARRAY[1..16] OF REAL;
    VI_Zone_Valve_States        : ARRAY[1..GVL_CONSTANTS.C_MAX_HEATING_CIRCUITS] OF BOOL;
    VI_Manifold_Pressures       : ARRAY[1..GVL_CONSTANTS.C_MAX_MANIFOLDS] OF REAL;
    VI_Manifold_Pump_States     : ARRAY[1..GVL_CONSTANTS.C_MAX_MANIFOLDS] OF BOOL;
    VI_Lighting_Base_Levels     : ARRAY[1..32] OF BYTE;
    VI_Socket_States            : ARRAY[1..GVL_CONSTANTS.C_MAX_SOCKETS] OF BOOL;
    VI_Blinds_Positions         : ARRAY[1..GVL_CONSTANTS.C_MAX_BLINDS] OF BYTE;
    VI_Allowed_IPs              : ARRAY[1..GVL_CONSTANTS.C_MAX_ALLOWED_IPS] OF STRING(15);
END_VAR

VAR_OUTPUT
    VO_Modbus_Registers         : ARRAY[0..GVL_CONSTANTS.C_MAX_MODBUS_REGISTERS-1] OF WORD;
    VO_Lighting_Override        : ARRAY[1..32] OF BYTE;
    VO_Blinds_Override          : ARRAY[1..GVL_CONSTANTS.C_MAX_BLINDS] OF BYTE;
    VO_Socket_Override          : ARRAY[1..GVL_CONSTANTS.C_MAX_SOCKETS] OF BOOL;
    VO_Arm_Req                  : BOOL;
    VO_Disarm_Req               : BOOL;
    VO_PIN_Code                 : STRING(4);
    VO_RFID_Tag                 : STRING(20);
    VO_2FA_Code_In              : STRING(6);
    VO_Data_Ready               : BOOL;
    VO_HMI_Status_Message       : STRING(200);
    VO_Telegram_Msg             : STRING(200);
    VO_Send_Telegram            : BOOL;
    VO_Set_Scenario_Req         : BOOL;
    VO_Target_Scenario          : E_SCENARIO_TYPE;
    VO_Set_Temp_Req             : BOOL;
    VO_Target_Zone              : INT;
    VO_Target_Temp              : REAL;
    VO_Set_Vent_Req             : BOOL;
    VO_Target_Vent_Speed        : BYTE;
    VO_Reset_Errors_Req         : BOOL;
    VO_Set_Config_Req           : BOOL;
    VO_Sync_Time_Req            : BOOL;
    VO_New_Time_MS              : UDINT;
END_VAR

VAR
    L_last_update_time          : UDINT;
    L_i                         : INT;
    L_j                         : INT;
    L_idx                       : INT;
    L_tmp_word                  : WORD;
    L_Code_UDINT                : UDINT;
    L_Prev_Fire                 : BOOL;
    L_Prev_Gas                  : BOOL;
    L_Prev_Flood                : BOOL;
    L_Prev_Security             : BOOL;
    L_Deduplicator              : FB_Command_Deduplication;
    L_CRC_Calc                  : FB_CRC32_Calculator;
    L_Calculated_CRC            : DWORD;
    L_IP_Allowed                : BOOL;
    L_Process_Command           : ST_Gateway_Command;
    L_Has_Command_To_Process    : BOOL;
END_VAR

VAR RETAIN
    L_Command_Buffer            : ARRAY[1..GVL_CONSTANTS.C_MAX_GATEWAY_COMMANDS] OF ST_Gateway_Command;
    L_Buffer_Head               : INT := 1;
    L_Buffer_Tail               : INT := 1;
    L_Buffer_Count              : INT := 0;
END_VAR

VO_Send_Telegram := FALSE;
IF VI_Fire_Alarm_Active AND NOT L_Prev_Fire THEN
    VO_Telegram_Msg := 'ВНИМАНИЕ! ПОЖАРНАЯ ТРЕВОГА!';
    VO_Send_Telegram := TRUE;
END_IF;
IF VI_Gas_Alarm_Active AND NOT L_Prev_Gas THEN
    VO_Telegram_Msg := 'ВНИМАНИЕ! УТЕЧКА ГАЗА!';
    VO_Send_Telegram := TRUE;
END_IF;
IF VI_Flood_Alarm_Active AND NOT L_Prev_Flood THEN
    VO_Telegram_Msg := 'ВНИМАНИЕ! ПРОТЕЧКА ВОДЫ!';
    VO_Send_Telegram := TRUE;
END_IF;
IF VI_Security_Armed AND NOT L_Prev_Security THEN
    VO_Telegram_Msg := 'ОХРАНА ВКЛЮЧЕНА';
    VO_Send_Telegram := TRUE;
ELSIF NOT VI_Security_Armed AND L_Prev_Security THEN
    VO_Telegram_Msg := 'ОХРАНА ОТКЛЮЧЕНА';
    VO_Send_Telegram := TRUE;
END_IF;

L_Prev_Fire := VI_Fire_Alarm_Active;
L_Prev_Gas := VI_Gas_Alarm_Active;
L_Prev_Flood := VI_Flood_Alarm_Active;
L_Prev_Security := VI_Security_Armed;

IF (VI_System_Time_MS - L_last_update_time) >= GVL_CONSTANTS.C_MS_IN_SECOND THEN
    L_last_update_time := VI_System_Time_MS;

    L_tmp_word := 0;
    IF VI_Local_PLC_Role = E_PLC_ROLE.ROLE_ACTIVE THEN L_tmp_word := L_tmp_word OR 1; END_IF;
    IF VI_Security_Armed THEN L_tmp_word := L_tmp_word OR 2; END_IF;
    IF VI_Flood_Alarm_Active THEN L_tmp_word := L_tmp_word OR 4; END_IF;
    IF VI_Gas_Alarm_Active THEN L_tmp_word := L_tmp_word OR 8; END_IF;
    IF VI_Fire_Alarm_Active THEN L_tmp_word := L_tmp_word OR 16; END_IF;
    VO_Modbus_Registers[0] := L_tmp_word;

    FOR L_i := 1 TO GVL_CONSTANTS.C_MAX_HEATING_CIRCUITS DO
        VO_Modbus_Registers[L_i] := TO_WORD(TO_INT(VI_FloorHeating_Temps[L_i] * REAL#10.0));
    END_FOR;

    FOR L_i := 1 TO 16 DO
        VO_Modbus_Registers[16 + L_i] := TO_WORD(TO_INT(VI_Room_Temps[L_i] * REAL#10.0));
    END_FOR;

    L_tmp_word := 0;
    FOR L_i := 1 TO GVL_CONSTANTS.C_MAX_HEATING_CIRCUITS DO
        IF VI_Zone_Valve_States[L_i] THEN
            L_tmp_word := L_tmp_word OR SHL(TO_WORD(1), L_i - 1);
        END_IF;
    END_FOR;
    VO_Modbus_Registers[33] := L_tmp_word;

    FOR L_i := 1 TO GVL_CONSTANTS.C_MAX_MANIFOLDS DO
        VO_Modbus_Registers[33 + L_i] := TO_WORD(TO_INT(VI_Manifold_Pressures[L_i] * REAL#100.0));
    END_FOR;

    FOR L_i := 1 TO 32 DO
        VO_Modbus_Registers[39 + L_i] := TO_WORD(VI_Lighting_Base_Levels[L_i]);
    END_FOR;

    FOR L_i := 1 TO GVL_CONSTANTS.C_MAX_BLINDS DO
        VO_Modbus_Registers[71 + L_i] := TO_WORD(VI_Blinds_Positions[L_i]);
    END_FOR;

    FOR L_i := 0 TO (GVL_CONSTANTS.C_MAX_SOCKETS - 1) / 16 DO
        L_tmp_word := 0;
        FOR L_j := 1 TO 16 DO
            L_idx := (L_i * 16) + L_j;
            IF L_idx <= GVL_CONSTANTS.C_MAX_SOCKETS THEN
                IF VI_Socket_States[L_idx] THEN
                    L_tmp_word := L_tmp_word OR SHL(TO_WORD(1), L_j - 1);
                END_IF;
            END_IF;
        END_FOR;
        VO_Modbus_Registers[92 + L_i] := L_tmp_word;
    END_FOR;

    VO_Modbus_Registers[100] := SEL(VI_Send_2FA_Req, 0, 1);
    IF VI_Send_2FA_Req THEN
        L_Code_UDINT := STRING_TO_UDINT(VI_2FA_Code);
        VO_Modbus_Registers[101] := TO_WORD(L_Code_UDINT AND 16#FFFF);
        VO_Modbus_Registers[102] := TO_WORD(SHR(L_Code_UDINT, 16));
    ELSE
        VO_Modbus_Registers[101] := 0;
        VO_Modbus_Registers[102] := 0;
    END_IF;

    VO_Data_Ready := TRUE;
END_IF;

VO_Arm_Req := FALSE;
VO_Disarm_Req := FALSE;
VO_Set_Scenario_Req := FALSE;
VO_Set_Temp_Req := FALSE;
VO_Set_Vent_Req := FALSE;
VO_Reset_Errors_Req := FALSE;
VO_Set_Config_Req := FALSE;
VO_Sync_Time_Req := FALSE;
L_Has_Command_To_Process := FALSE;

IF VI_Command_Received THEN
    IF VI_Local_PLC_Role = E_PLC_ROLE.ROLE_ACTIVE THEN
        L_Process_Command := VI_Incoming_Command;
        L_Has_Command_To_Process := TRUE;
    ELSE
        IF L_Buffer_Count < GVL_CONSTANTS.C_MAX_GATEWAY_COMMANDS THEN
            L_Command_Buffer[L_Buffer_Head] := VI_Incoming_Command;
            L_Buffer_Head := L_Buffer_Head + 1;
            IF L_Buffer_Head > GVL_CONSTANTS.C_MAX_GATEWAY_COMMANDS THEN L_Buffer_Head := 1; END_IF;
            L_Buffer_Count := L_Buffer_Count + 1;
        END_IF;
    END_IF;
END_IF;

IF NOT L_Has_Command_To_Process AND (VI_Local_PLC_Role = E_PLC_ROLE.ROLE_ACTIVE) AND (L_Buffer_Count > 0) THEN
    L_Process_Command := L_Command_Buffer[L_Buffer_Tail];
    L_Buffer_Tail := L_Buffer_Tail + 1;
    IF L_Buffer_Tail > GVL_CONSTANTS.C_MAX_GATEWAY_COMMANDS THEN L_Buffer_Tail := 1; END_IF;
    L_Buffer_Count := L_Buffer_Count - 1;
    L_Has_Command_To_Process := TRUE;
END_IF;

IF L_Has_Command_To_Process THEN
    L_IP_Allowed := FALSE;
    IF L_Process_Command.source_ip = '' THEN
        L_IP_Allowed := TRUE;
    ELSE
        FOR L_i := 1 TO GVL_CONSTANTS.C_MAX_ALLOWED_IPS DO
            IF VI_Allowed_IPs[L_i] = L_Process_Command.source_ip THEN
                L_IP_Allowed := TRUE;
                EXIT;
            END_IF;
        END_FOR;
    END_IF;

    IF NOT L_IP_Allowed THEN
        VO_HMI_Status_Message := 'Gateway: Ошибка безопасности (Неизвестный IP)';
        RETURN;
    END_IF;

    L_CRC_Calc();
    L_Calculated_CRC := L_CRC_Calc.VO_CRC;

    IF L_Calculated_CRC = L_Process_Command.crc32 THEN
        L_Deduplicator(
            VI_Command_ID := L_Process_Command.command_id,
            VI_Command_Type := L_Process_Command.command_type,
            VI_Command_Value := L_Process_Command.target_value,
            VI_System_Time_MS := VI_System_Time_MS
        );

        IF L_Deduplicator.VO_Is_New_Command THEN
            CASE L_Process_Command.command_type OF
                E_Gateway_Command_Type.CMD_SET_SCENARIO:
                    VO_Set_Scenario_Req := TRUE;
                    VO_Target_Scenario := L_Process_Command.target_scenario;
                    VO_HMI_Status_Message := 'Gateway: Сценарий изменен';
                E_Gateway_Command_Type.CMD_SET_LIGHT:
                    IF (L_Process_Command.target_zone >= 1) AND (L_Process_Command.target_zone <= 32) THEN
                        VO_Lighting_Override[L_Process_Command.target_zone] := TO_BYTE(L_Process_Command.target_value);
                        VO_HMI_Status_Message := 'Gateway: Команда освещения принята';
                    END_IF;
                E_Gateway_Command_Type.CMD_SET_BLINDS:
                    IF (L_Process_Command.target_zone >= 1) AND (L_Process_Command.target_zone <= GVL_CONSTANTS.C_MAX_BLINDS) THEN
                        VO_Blinds_Override[L_Process_Command.target_zone] := TO_BYTE(L_Process_Command.target_value);
                        VO_HMI_Status_Message := 'Gateway: Команда штор принята';
                    END_IF;
                E_Gateway_Command_Type.CMD_SET_SOCKET:
                    IF (L_Process_Command.target_zone >= 1) AND (L_Process_Command.target_zone <= GVL_CONSTANTS.C_MAX_SOCKETS) THEN
                        VO_Socket_Override[L_Process_Command.target_zone] := L_Process_Command.target_on_off;
                        VO_HMI_Status_Message := 'Gateway: Команда розетки принята';
                    END_IF;
                E_Gateway_Command_Type.CMD_SET_SECURITY:
                    IF L_Process_Command.target_armed THEN
                        VO_Arm_Req := TRUE;
                    ELSE
                        VO_Disarm_Req := TRUE;
                    END_IF;
                    VO_PIN_Code := L_Process_Command.target_pin;
                    VO_2FA_Code_In := L_Process_Command.target_2fa_code;
                    VO_HMI_Status_Message := 'Gateway: Запрос охраны принят';
                E_Gateway_Command_Type.CMD_SET_TEMP:
                    IF (L_Process_Command.target_zone >= 1) AND (L_Process_Command.target_zone <= GVL_CONSTANTS.C_MAX_HEATING_CIRCUITS) THEN
                        VO_Set_Temp_Req := TRUE;
                        VO_Target_Zone := L_Process_Command.target_zone;
                        VO_Target_Temp := L_Process_Command.target_value;
                        VO_HMI_Status_Message := 'Gateway: Уставка температуры изменена';
                    END_IF;
                E_Gateway_Command_Type.CMD_SET_VENT:
                    VO_Set_Vent_Req := TRUE;
                    VO_Target_Vent_Speed := TO_BYTE(L_Process_Command.target_value);
                    VO_HMI_Status_Message := 'Gateway: Уставка вентиляции изменена';
                E_Gateway_Command_Type.CMD_TELEGRAM_MSG:
                    VO_Telegram_Msg := L_Process_Command.telegram_msg;
                    VO_Send_Telegram := TRUE;
                    VO_HMI_Status_Message := 'Gateway: Сообщение Telegram отправлено';
                E_Gateway_Command_Type.CMD_SYNC_TIME:
                    VO_Sync_Time_Req := TRUE;
                    VO_New_Time_MS := REAL_TO_UDINT(L_Process_Command.target_value);
                    VO_HMI_Status_Message := 'Gateway: Время синхронизировано';
                E_Gateway_Command_Type.CMD_RESET_ERRORS:
                    VO_Reset_Errors_Req := TRUE;
                    VO_HMI_Status_Message := 'Gateway: Запрос на сброс ошибок принят';
                E_Gateway_Command_Type.CMD_SET_CONFIG:
                    VO_Set_Config_Req := TRUE;
                    VO_HMI_Status_Message := 'Gateway: Запрос на применение конфигурации принят';
            END_CASE;
        END_IF;
    ELSE
        VO_HMI_Status_Message := 'Gateway: Ошибка CRC команды';
    END_IF;
END_IF;

// >>> BULK_SYNC_ANCHOR: FB_Gateway_Interface <<<
END_FUNCTION_BLOCK

(* ---- FB_Heating_Adapter_CopyOut.st ---- *)
FUNCTION_BLOCK FB_Heating_Adapter_CopyOut
VAR_INPUT
    VI_Zone_Valves : ARRAY[1..GVL_CONSTANTS.C_MAX_HEATING_CIRCUITS] OF BOOL;
END_VAR
VAR_IN_OUT
    VIO_Zone_Valves_State : ARRAY[1..GVL_CONSTANTS.C_MAX_HEATING_CIRCUITS] OF BOOL;
END_VAR
VAR
    L_i : INT;
END_VAR

// Extracted candidate from PRG_Heating S6.
// Not connected yet.
// No global switching yet.

FOR L_i := 1 TO GVL_CONSTANTS.C_MAX_HEATING_CIRCUITS DO
    VIO_Zone_Valves_State[L_i] := VI_Zone_Valves[L_i];
END_FOR;

END_FUNCTION_BLOCK
// >>> BULK_SYNC_ANCHOR: FB_Heating_Adapter_CopyOut <<<
